LIN {X 0,Y 426.381,Z 386.373,A -85,B 0,C 180,E1 -9911.885,E2 -9911.885} C_VEL
LIN {X 0,Y 426.7,Z 374.582,A -85,B 0,C 180,E1 -9912.449,E2 -9912.449} C_VEL
LIN {X 0,Y 426.837,Z 364.477,A -85,B 0,C 180,E1 -9912.777,E2 -9912.777} C_VEL
LIN {X 0,Y 427.571,Z 302.941,A -85,B 0,C 180,E1 -9914.039,E2 -9914.039} C_VEL
LIN {X 0,Y 425.288,Z 288.443,A -85,B 0,C 180,E1 -9914.407,E2 -9914.407} C_VEL
LIN {X 0,Y 425.647,Z 277.739,A -85,B 0,C 180,E1 -9917.284,E2 -9917.284} C_VEL
LIN {X 0,Y 425.385,Z 272.31,A -85,B 0,C 180,E1 -9918.851,E2 -9918.851} C_VEL
LIN {X 0,Y 425.275,Z 272.323,A -85,B 0,C 180,E1 -9922.333,E2 -9922.333} C_VEL
LIN {X 0,Y 425.247,Z 272.327,A -85,B 0,C 180,E1 -9925.442,E2 -9925.442} C_VEL
LIN {X 0,Y 425.282,Z 272.324,A -85,B 0,C 180,E1 -9928.852,E2 -9928.852} C_VEL
LIN {X 0,Y 425.243,Z 272.328,A -85,B 0,C 180,E1 -9931.921,E2 -9931.921} C_VEL
LIN {X 0,Y 425.274,Z 272.323,A -85,B 0,C 180,E1 -9935.33,E2 -9935.33} C_VEL
LIN {X 0,Y 425.253,Z 272.327,A -85,B 0,C 180,E1 -9938.895,E2 -9938.895} C_VEL
LIN {X 0,Y 425.252,Z 272.326,A -85,B 0,C 180,E1 -9941.951,E2 -9941.951} C_VEL
LIN {X 0,Y 425.252,Z 272.328,A -85,B 0,C 180,E1 -9945.277,E2 -9945.277} C_VEL
LIN {X 0,Y 425.238,Z 272.327,A -85,B 0,C 180,E1 -9948.616,E2 -9948.616} C_VEL
LIN {X 0,Y 425.254,Z 272.326,A -85,B 0,C 180,E1 -9951.095,E2 -9951.095} C_VEL
LIN {X 0,Y 425.259,Z 272.325,A -85,B 0,C 180,E1 -9954.659,E2 -9954.659} C_VEL
LIN {X 0,Y 425.221,Z 272.329,A -85,B 0,C 180,E1 -9958.068,E2 -9958.068} C_VEL
LIN {X 0,Y 425.285,Z 272.322,A -85,B 0,C 180,E1 -9961.363,E2 -9961.363} C_VEL
LIN {X 0,Y 425.248,Z 272.327,A -85,B 0,C 180,E1 -9964.55,E2 -9964.55} C_VEL
LIN {X 0,Y 425.238,Z 272.328,A -85,B 0,C 180,E1 -9967.657,E2 -9967.657} C_VEL
LIN {X 0,Y 425.31,Z 272.319,A -85,B 0,C 180,E1 -9970.7,E2 -9970.7} C_VEL
LIN {X 0,Y 425.335,Z 272.316,A -85,B 0,C 180,E1 -9973.685,E2 -9973.685} C_VEL
LIN {X 0,Y 425.377,Z 272.31,A -85,B 0,C 180,E1 -9977.596,E2 -9977.596} C_VEL
LIN {X 0,Y 425.387,Z 272.309,A -85,B 0,C 180,E1 -9981.447,E2 -9981.447} C_VEL
LIN {X 0,Y 425.52,Z 272.295,A -85,B 0,C 180,E1 -9984.311,E2 -9984.311} C_VEL
LIN {X 0,Y 425.334,Z 272.315,A -85,B 0,C 180,E1 -9986.427,E2 -9986.427} C_VEL
LIN {X 0,Y 424.809,Z 272.381,A -85,B 0,C 180,E1 -9987.218,E2 -9987.218} C_VEL
LIN {X 0,Y 422.102,Z 272.72,A -85,B 0,C 180,E1 -9988.506,E2 -9988.506} C_VEL
LIN {X 0,Y 419.705,Z 273.017,A -85,B 0,C 180,E1 -9989.545,E2 -9989.545} C_VEL
LIN {X 0,Y 418.62,Z 273.153,A -85,B 0,C 180,E1 -9990.347,E2 -9990.347} C_VEL
LIN {X 0,Y 418.506,Z 273.164,A -85,B 0,C 180,E1 -9990.619,E2 -9990.619} C_VEL
LIN {X 0,Y 418.461,Z 273.172,A -85,B 0,C 180,E1 -9992.886,E2 -9992.886} C_VEL
LIN {X 0,Y 418.436,Z 273.176,A -85,B 0,C 180,E1 -9996.75,E2 -9996.75} C_VEL
LIN {X 0,Y 418.304,Z 273.192,A -85,B 0,C 180,E1 -9999.67,E2 -9999.67} C_VEL
LIN {X 0,Y 418.296,Z 273.193,A -85,B 0,C 180,E1 -10003.006,E2 -10003.006} C_VEL
LIN {X 0,Y 418.253,Z 273.199,A -85,B 0,C 180,E1 -10006.735,E2 -10006.735} C_VEL
LIN {X 0,Y 418.211,Z 273.203,A -85,B 0,C 180,E1 -10009.791,E2 -10009.791} C_VEL
LIN {X 0,Y 418.18,Z 273.207,A -85,B 0,C 180,E1 -10012.737,E2 -10012.737} C_VEL
LIN {X 0,Y 418.216,Z 273.202,A -85,B 0,C 180,E1 -10015.905,E2 -10015.905} C_VEL
LIN {X 0,Y 418.218,Z 273.204,A -85,B 0,C 180,E1 -10019.163,E2 -10019.163} C_VEL
LIN {X 0,Y 418.202,Z 273.204,A -85,B 0,C 180,E1 -10022.846,E2 -10022.846} C_VEL
LIN {X 0,Y 418.195,Z 273.205,A -85,B 0,C 180,E1 -10026.241,E2 -10026.241} C_VEL
LIN {X 0,Y 418.217,Z 273.203,A -85,B 0,C 180,E1 -10029.683,E2 -10029.683} C_VEL
LIN {X 0,Y 418.235,Z 273.2,A -85,B 0,C 180,E1 -10032.333,E2 -10032.333} C_VEL
LIN {X 0,Y 418.226,Z 273.201,A -85,B 0,C 180,E1 -10035.117,E2 -10035.117} C_VEL
LIN {X 0,Y 418.246,Z 273.201,A -85,B 0,C 180,E1 -10037.777,E2 -10037.777} C_VEL
LIN {X 0,Y 418.221,Z 273.202,A -85,B 0,C 180,E1 -10041.564,E2 -10041.564} C_VEL
LIN {X 0,Y 418.218,Z 273.202,A -85,B 0,C 180,E1 -10045.163,E2 -10045.163} C_VEL
LIN {X 0,Y 418.205,Z 273.203,A -85,B 0,C 180,E1 -10047.476,E2 -10047.476} C_VEL
LIN {X 0,Y 418.231,Z 273.2,A -85,B 0,C 180,E1 -10050.9,E2 -10050.9} C_VEL
LIN {X 0,Y 418.225,Z 273.203,A -85,B 0,C 180,E1 -10054.1,E2 -10054.1} C_VEL
LIN {X 0,Y 418.198,Z 273.205,A -85,B 0,C 180,E1 -10057.268,E2 -10057.268} C_VEL
LIN {X 0,Y 418.252,Z 273.2,A -85,B 0,C 180,E1 -10060.369,E2 -10060.369} C_VEL
LIN {X 0,Y 418.287,Z 273.194,A -85,B 0,C 180,E1 -10063.409,E2 -10063.409} C_VEL
LIN {X 0,Y 418.32,Z 273.189,A -85,B 0,C 180,E1 -10067.004,E2 -10067.004} C_VEL
LIN {X 0,Y 418.313,Z 273.191,A -85,B 0,C 180,E1 -10070.333,E2 -10070.333} C_VEL
LIN {X 0,Y 418.446,Z 273.173,A -85,B 0,C 180,E1 -10073.253,E2 -10073.253} C_VEL
LIN {X 0,Y 418.303,Z 273.191,A -85,B 0,C 180,E1 -10075.186,E2 -10075.186} C_VEL
LIN {X 0,Y 418.516,Z 273.165,A -85,B 0,C 180,E1 -10078.08,E2 -10078.08} C_VEL
LIN {X 0,Y 418.526,Z 273.164,A -85,B 0,C 180,E1 -10080.005,E2 -10080.005} C_VEL
LIN {X 0,Y 418.474,Z 273.172,A -85,B 0,C 180,E1 -10082.893,E2 -10082.893} C_VEL
LIN {X 0,Y 418.473,Z 273.17,A -85,B 0,C 180,E1 -10085.788,E2 -10085.788} C_VEL
LIN {X 0,Y 418.364,Z 273.184,A -85,B 0,C 180,E1 -10088.7,E2 -10088.7} C_VEL
LIN {X 0,Y 418.302,Z 273.191,A -85,B 0,C 180,E1 -10091.636,E2 -10091.636} C_VEL
LIN {X 0,Y 418.268,Z 273.196,A -85,B 0,C 180,E1 -10094.602,E2 -10094.602} C_VEL
LIN {X 0,Y 418.247,Z 273.199,A -85,B 0,C 180,E1 -10097.61,E2 -10097.61} C_VEL
LIN {X 0,Y 418.242,Z 273.199,A -85,B 0,C 180,E1 -10100.667,E2 -10100.667} C_VEL
LIN {X 0,Y 418.25,Z 273.199,A -85,B 0,C 180,E1 -10103.787,E2 -10103.787} C_VEL
LIN {X 0,Y 418.219,Z 273.202,A -85,B 0,C 180,E1 -10107.051,E2 -10107.051} C_VEL
LIN {X 0,Y 418.238,Z 273.199,A -85,B 0,C 180,E1 -10110.276,E2 -10110.276} C_VEL
LIN {X 0,Y 418.229,Z 273.202,A -85,B 0,C 180,E1 -10113.683,E2 -10113.683} C_VEL
LIN {X 0,Y 418.231,Z 273.2,A -85,B 0,C 180,E1 -10117.229,E2 -10117.229} C_VEL
LIN {X 0,Y 418.206,Z 273.203,A -85,B 0,C 180,E1 -10120.87,E2 -10120.87} C_VEL
LIN {X 0,Y 418.202,Z 273.204,A -85,B 0,C 180,E1 -10123.731,E2 -10123.731} C_VEL
LIN {X 0,Y 418.198,Z 273.205,A -85,B 0,C 180,E1 -10126.45,E2 -10126.45} C_VEL
LIN {X 0,Y 418.208,Z 273.203,A -85,B 0,C 180,E1 -10129.136,E2 -10129.136} C_VEL
LIN {X 0,Y 418.238,Z 273.199,A -85,B 0,C 180,E1 -10132.778,E2 -10132.778} C_VEL
LIN {X 0,Y 418.235,Z 273.202,A -85,B 0,C 180,E1 -10136.324,E2 -10136.324} C_VEL
LIN {X 0,Y 418.242,Z 273.199,A -85,B 0,C 180,E1 -10139.73,E2 -10139.73} C_VEL
LIN {X 0,Y 418.205,Z 273.203,A -85,B 0,C 180,E1 -10143.018,E2 -10143.018} C_VEL
LIN {X 0,Y 418.321,Z 273.357,A -85,B 0,C 180,E1 -10144.988,E2 -10144.988} C_VEL
LIN {X 0,Y 419.897,Z 283.23,A -85,B 0,C 180,E1 -10147.361,E2 -10147.361} C_VEL
LIN {X 0,Y 419.321,Z 295.276,A -85,B 0,C 180,E1 -10150.104,E2 -10150.104} C_VEL
LIN {X 0,Y 418.425,Z 312.199,A -85,B 0,C 180,E1 -10153.912,E2 -10153.912} C_VEL
LIN {X 0,Y 418.146,Z 318.839,A -85,B 0,C 180,E1 -10155.399,E2 -10155.399} C_VEL
LIN {X 0,Y 420.457,Z 340.768,A -85,B 0,C 180,E1 -10155.935,E2 -10155.935} C_VEL
LIN {X 0,Y 419.749,Z 397.826,A -85,B 0,C 180,E1 -10157.153,E2 -10157.153} C_VEL
LIN {X 0,Y 419.378,Z 409.923,A -85,B 0,C 180,E1 -10157.603,E2 -10157.603} C_VEL
LIN {X 0,Y 418.995,Z 419.778,A -85,B 0,C 180,E1 -10158.145,E2 -10158.145} C_VEL
LIN {X 0,Y 418.642,Z 428.317,A -85,B 0,C 180,E1 -10158.748,E2 -10158.748} C_VEL
LIN {X 0,Y 418.327,Z 436.579,A -85,B 0,C 180,E1 -10159.475,E2 -10159.475} C_VEL
LIN {X 0,Y 418.04,Z 444.456,A -85,B 0,C 180,E1 -10160.323,E2 -10160.323} C_VEL
LIN {X 0,Y 417.61,Z 453.524,A -85,B 0,C 180,E1 -10161.534,E2 -10161.534} C_VEL
LIN {X 0,Y 417.386,Z 460.516,A -85,B 0,C 180,E1 -10162.747,E2 -10162.747} C_VEL
LIN {X 0,Y 417.15,Z 466.408,A -85,B 0,C 180,E1 -10164.037,E2 -10164.037} C_VEL
LIN {X 0,Y 417.164,Z 470.478,A -85,B 0,C 180,E1 -10165.17,E2 -10165.17} C_VEL
LIN {X 0,Y 417.047,Z 473.209,A -85,B 0,C 180,E1 -10166.137,E2 -10166.137} C_VEL
LIN {X 0,Y 417.079,Z 475.349,A -85,B 0,C 180,E1 -10167.104,E2 -10167.104} C_VEL
LIN {X 0,Y 417.078,Z 476.927,A -85,B 0,C 180,E1 -10168.07,E2 -10168.07} C_VEL
LIN {X 0,Y 417.036,Z 477.901,A -85,B 0,C 180,E1 -10169.036,E2 -10169.036} C_VEL
LIN {X 0,Y 417.031,Z 478.279,A -85,B 0,C 180,E1 -10170.002,E2 -10170.002} C_VEL
LIN {X 0,Y 417.017,Z 478.147,A -85,B 0,C 180,E1 -10170.967,E2 -10170.967} C_VEL
LIN {X 0,Y 417.075,Z 477.507,A -85,B 0,C 180,E1 -10171.933,E2 -10171.933} C_VEL
LIN {X 0,Y 417.042,Z 476.345,A -85,B 0,C 180,E1 -10172.899,E2 -10172.899} C_VEL
LIN {X 0,Y 417.087,Z 473.43,A -85,B 0,C 180,E1 -10174.35,E2 -10174.35} C_VEL
LIN {X 0,Y 417.179,Z 469.185,A -85,B 0,C 180,E1 -10175.803,E2 -10175.803} C_VEL
LIN {X 0,Y 417.447,Z 463.483,A -85,B 0,C 180,E1 -10177.256,E2 -10177.256} C_VEL
LIN {X 0,Y 417.721,Z 457.262,A -85,B 0,C 180,E1 -10178.467,E2 -10178.467} C_VEL
LIN {X 0,Y 418.11,Z 451.182,A -85,B 0,C 180,E1 -10179.434,E2 -10179.434} C_VEL
LIN {X 0,Y 418.569,Z 443.809,A -85,B 0,C 180,E1 -10180.4,E2 -10180.4} C_VEL
LIN {X 0,Y 418.977,Z 435.985,A -85,B 0,C 180,E1 -10181.246,E2 -10181.246} C_VEL
LIN {X 0,Y 419.352,Z 429.321,A -85,B 0,C 180,E1 -10181.849,E2 -10181.849} C_VEL
LIN {X 0,Y 419.749,Z 421.293,A -85,B 0,C 180,E1 -10182.45,E2 -10182.45} C_VEL
LIN {X 0,Y 420.179,Z 412.209,A -85,B 0,C 180,E1 -10182.99,E2 -10182.99} C_VEL
LIN {X 0,Y 420.662,Z 402.136,A -85,B 0,C 180,E1 -10183.436,E2 -10183.436} C_VEL
LIN {X 0,Y 421.087,Z 390.096,A -85,B 0,C 180,E1 -10183.789,E2 -10183.789} C_VEL
LIN {X 0,Y 421.982,Z 339.107,A -85,B 0,C 180,E1 -10184.931,E2 -10184.931} C_VEL
LIN {X 0,Y 420.236,Z 325.232,A -85,B 0,C 180,E1 -10185.362,E2 -10185.362} C_VEL
LIN {X 0,Y 418.562,Z 315.696,A -85,B 0,C 180,E1 -10185.71,E2 -10185.71} C_VEL
LIN {X 0,Y 419.082,Z 299.8,A -85,B 0,C 180,E1 -10188.835,E2 -10188.835} C_VEL
LIN {X 0,Y 419.665,Z 282.928,A -85,B 0,C 180,E1 -10192.137,E2 -10192.137} C_VEL
LIN {X 0,Y 419.287,Z 277.639,A -85,B 0,C 180,E1 -10193.214,E2 -10193.214} C_VEL
LIN {X 0,Y 418.303,Z 273.195,A -85,B 0,C 180,E1 -10194.177,E2 -10194.177} C_VEL
LIN {X 0,Y 418.212,Z 273.208,A -85,B 0,C 180,E1 -10198.07,E2 -10198.07} C_VEL
LIN {X 0,Y 418.221,Z 273.206,A -85,B 0,C 180,E1 -10201.011,E2 -10201.011} C_VEL
LIN {X 0,Y 418.205,Z 273.204,A -85,B 0,C 180,E1 -10203.682,E2 -10203.682} C_VEL
LIN {X 0,Y 418.238,Z 273.201,A -85,B 0,C 180,E1 -10207.226,E2 -10207.226} C_VEL
LIN {X 0,Y 418.222,Z 273.205,A -85,B 0,C 180,E1 -10210.949,E2 -10210.949} C_VEL
LIN {X 0,Y 418.195,Z 273.202,A -85,B 0,C 180,E1 -10213.724,E2 -10213.724} C_VEL
LIN {X 0,Y 418.193,Z 273.203,A -85,B 0,C 180,E1 -10216.443,E2 -10216.443} C_VEL
LIN {X 0,Y 418.224,Z 273.201,A -85,B 0,C 180,E1 -10219.132,E2 -10219.132} C_VEL
LIN {X 0,Y 418.253,Z 273.197,A -85,B 0,C 180,E1 -10222.774,E2 -10222.774} C_VEL
LIN {X 0,Y 418.249,Z 273.196,A -85,B 0,C 180,E1 -10226.319,E2 -10226.319} C_VEL
LIN {X 0,Y 418.258,Z 273.198,A -85,B 0,C 180,E1 -10229.725,E2 -10229.725} C_VEL
LIN {X 0,Y 418.24,Z 273.204,A -85,B 0,C 180,E1 -10233.015,E2 -10233.015} C_VEL
LIN {X 0,Y 418.289,Z 273.196,A -85,B 0,C 180,E1 -10236.215,E2 -10236.215} C_VEL
LIN {X 0,Y 418.265,Z 273.199,A -85,B 0,C 180,E1 -10239.334,E2 -10239.334} C_VEL
LIN {X 0,Y 418.401,Z 273.384,A -85,B 0,C 180,E1 -10242.145,E2 -10242.145} C_VEL
LIN {X 0,Y 419.951,Z 279.942,A -85,B 0,C 180,E1 -10243.28,E2 -10243.28} C_VEL
LIN {X 0,Y 419.768,Z 287.188,A -85,B 0,C 180,E1 -10244.38,E2 -10244.38} C_VEL
LIN {X 0,Y 422.411,Z 302.684,A -85,B 0,C 180,E1 -10244.912,E2 -10244.912} C_VEL
LIN {X 0,Y 421.611,Z 349.13,A -85,B 0,C 180,E1 -10245.985,E2 -10245.985} C_VEL
LIN {X 0,Y 421.112,Z 370.004,A -85,B 0,C 180,E1 -10246.484,E2 -10246.484} C_VEL
LIN {X 0,Y 420.721,Z 381.477,A -85,B 0,C 180,E1 -10246.963,E2 -10246.963} C_VEL
LIN {X 0,Y 420.384,Z 389.953,A -85,B 0,C 180,E1 -10247.443,E2 -10247.443} C_VEL
LIN {X 0,Y 420.045,Z 398.323,A -85,B 0,C 180,E1 -10248.046,E2 -10248.046} C_VEL
LIN {X 0,Y 419.546,Z 406.458,A -85,B 0,C 180,E1 -10248.766,E2 -10248.766} C_VEL
LIN {X 0,Y 419.242,Z 414.199,A -85,B 0,C 180,E1 -10249.614,E2 -10249.614} C_VEL
LIN {X 0,Y 418.658,Z 423.145,A -85,B 0,C 180,E1 -10250.819,E2 -10250.819} C_VEL
LIN {X 0,Y 418.184,Z 430.047,A -85,B 0,C 180,E1 -10252.026,E2 -10252.026} C_VEL
LIN {X 0,Y 417.964,Z 435.543,A -85,B 0,C 180,E1 -10253.236,E2 -10253.236} C_VEL
LIN {X 0,Y 417.565,Z 439.126,A -85,B 0,C 180,E1 -10254.2,E2 -10254.2} C_VEL
LIN {X 0,Y 417.492,Z 443.184,A -85,B 0,C 180,E1 -10255.651,E2 -10255.651} C_VEL
LIN {X 0,Y 417.263,Z 445.971,A -85,B 0,C 180,E1 -10257.099,E2 -10257.099} C_VEL
LIN {X 0,Y 417.129,Z 447.063,A -85,B 0,C 180,E1 -10258.064,E2 -10258.064} C_VEL
LIN {X 0,Y 417.042,Z 447.644,A -85,B 0,C 180,E1 -10259.03,E2 -10259.03} C_VEL
LIN {X 0,Y 417.032,Z 447.72,A -85,B 0,C 180,E1 -10259.995,E2 -10259.995} C_VEL
LIN {X 0,Y 417.04,Z 447.28,A -85,B 0,C 180,E1 -10260.961,E2 -10260.961} C_VEL
LIN {X 0,Y 417.106,Z 446.234,A -85,B 0,C 180,E1 -10261.926,E2 -10261.926} C_VEL
LIN {X 0,Y 417.248,Z 443.672,A -85,B 0,C 180,E1 -10263.375,E2 -10263.375} C_VEL
LIN {X 0,Y 417.277,Z 439.705,A -85,B 0,C 180,E1 -10264.826,E2 -10264.826} C_VEL
LIN {X 0,Y 417.473,Z 434.89,A -85,B 0,C 180,E1 -10266.133,E2 -10266.133} C_VEL
LIN {X 0,Y 417.768,Z 428.599,A -85,B 0,C 180,E1 -10267.462,E2 -10267.462} C_VEL
LIN {X 0,Y 418.037,Z 421.038,A -85,B 0,C 180,E1 -10268.697,E2 -10268.697} C_VEL
LIN {X 0,Y 418.34,Z 413.649,A -85,B 0,C 180,E1 -10269.666,E2 -10269.666} C_VEL
LIN {X 0,Y 418.69,Z 405.785,A -85,B 0,C 180,E1 -10270.512,E2 -10270.512} C_VEL
LIN {X 0,Y 418.944,Z 397.53,A -85,B 0,C 180,E1 -10271.24,E2 -10271.24} C_VEL
LIN {X 0,Y 419.335,Z 387.148,A -85,B 0,C 180,E1 -10271.965,E2 -10271.965} C_VEL
LIN {X 0,Y 419.663,Z 375.717,A -85,B 0,C 180,E1 -10272.538,E2 -10272.538} C_VEL
LIN {X 0,Y 419.818,Z 366.071,A -85,B 0,C 180,E1 -10272.871,E2 -10272.871} C_VEL
LIN {X 0,Y 420.509,Z 303.025,A -85,B 0,C 180,E1 -10274.217,E2 -10274.217} C_VEL
LIN {X 0,Y 418.277,Z 288.664,A -85,B 0,C 180,E1 -10274.592,E2 -10274.592} C_VEL
LIN {X 0,Y 418.618,Z 277.685,A -85,B 0,C 180,E1 -10277.583,E2 -10277.583} C_VEL
LIN {X 0,Y 418.351,Z 273.186,A -85,B 0,C 180,E1 -10278.862,E2 -10278.862} C_VEL
LIN {X 0,Y 418.215,Z 273.203,A -85,B 0,C 180,E1 -10282.731,E2 -10282.731} C_VEL
LIN {X 0,Y 418.211,Z 273.203,A -85,B 0,C 180,E1 -10285.901,E2 -10285.901} C_VEL
LIN {X 0,Y 418.239,Z 273.199,A -85,B 0,C 180,E1 -10289.157,E2 -10289.157} C_VEL
LIN {X 0,Y 418.236,Z 273.202,A -85,B 0,C 180,E1 -10292.838,E2 -10292.838} C_VEL
LIN {X 0,Y 418.219,Z 273.202,A -85,B 0,C 180,E1 -10296.231,E2 -10296.231} C_VEL
LIN {X 0,Y 418.184,Z 273.206,A -85,B 0,C 180,E1 -10299.681,E2 -10299.681} C_VEL
LIN {X 0,Y 418.193,Z 273.206,A -85,B 0,C 180,E1 -10302.314,E2 -10302.314} C_VEL
LIN {X 0,Y 418.203,Z 273.205,A -85,B 0,C 180,E1 -10305.103,E2 -10305.103} C_VEL
LIN {X 0,Y 418.205,Z 273.203,A -85,B 0,C 180,E1 -10307.761,E2 -10307.761} C_VEL
LIN {X 0,Y 418.205,Z 273.204,A -85,B 0,C 180,E1 -10310.616,E2 -10310.616} C_VEL
LIN {X 0,Y 418.203,Z 273.203,A -85,B 0,C 180,E1 -10313.97,E2 -10313.97} C_VEL
LIN {X 0,Y 418.215,Z 273.202,A -85,B 0,C 180,E1 -10317.151,E2 -10317.151} C_VEL
LIN {X 0,Y 418.224,Z 273.202,A -85,B 0,C 180,E1 -10320.891,E2 -10320.891} C_VEL
LIN {X 0,Y 418.224,Z 273.201,A -85,B 0,C 180,E1 -10324.091,E2 -10324.091} C_VEL
LIN {X 0,Y 418.189,Z 273.206,A -85,B 0,C 180,E1 -10327.26,E2 -10327.26} C_VEL
LIN {X 0,Y 418.231,Z 273.2,A -85,B 0,C 180,E1 -10330.36,E2 -10330.36} C_VEL
LIN {X 0,Y 418.264,Z 273.196,A -85,B 0,C 180,E1 -10333.401,E2 -10333.401} C_VEL
LIN {X 0,Y 418.301,Z 273.192,A -85,B 0,C 180,E1 -10336.991,E2 -10336.991} C_VEL
LIN {X 0,Y 418.306,Z 273.192,A -85,B 0,C 180,E1 -10340.326,E2 -10340.326} C_VEL
LIN {X 0,Y 418.438,Z 273.176,A -85,B 0,C 180,E1 -10343.247,E2 -10343.247} C_VEL
LIN {X 0,Y 418.291,Z 273.193,A -85,B 0,C 180,E1 -10345.179,E2 -10345.179} C_VEL
LIN {X 0,Y 418.489,Z 273.169,A -85,B 0,C 180,E1 -10348.074,E2 -10348.074} C_VEL
LIN {X 0,Y 418.506,Z 273.164,A -85,B 0,C 180,E1 -10350.619,E2 -10350.619} C_VEL
LIN {X 0,Y 417.738,Z 273.263,A -85,B 0,C 180,E1 -10351.422,E2 -10351.422} C_VEL
LIN {X 0,Y 414.75,Z 273.634,A -85,B 0,C 180,E1 -10352.724,E2 -10352.724} C_VEL
LIN {X 0,Y 412.303,Z 273.939,A -85,B 0,C 180,E1 -10353.775,E2 -10353.775} C_VEL
LIN {X 0,Y 411.308,Z 274.064,A -85,B 0,C 180,E1 -10354.59,E2 -10354.59} C_VEL
LIN {X 0,Y 411.254,Z 274.069,A -85,B 0,C 180,E1 -10354.865,E2 -10354.865} C_VEL
LIN {X 0,Y 411.402,Z 274.051,A -85,B 0,C 180,E1 -10356.866,E2 -10356.866} C_VEL
LIN {X 0,Y 411.252,Z 274.071,A -85,B 0,C 180,E1 -10359.838,E2 -10359.838} C_VEL
LIN {X 0,Y 411.255,Z 274.069,A -85,B 0,C 180,E1 -10363.109,E2 -10363.109} C_VEL
LIN {X 0,Y 411.199,Z 274.078,A -85,B 0,C 180,E1 -10366.889,E2 -10366.889} C_VEL
LIN {X 0,Y 411.172,Z 274.08,A -85,B 0,C 180,E1 -10369.988,E2 -10369.988} C_VEL
LIN {X 0,Y 411.146,Z 274.084,A -85,B 0,C 180,E1 -10373.149,E2 -10373.149} C_VEL
LIN {X 0,Y 411.182,Z 274.079,A -85,B 0,C 180,E1 -10376.382,E2 -10376.382} C_VEL
LIN {X 0,Y 411.155,Z 274.081,A -85,B 0,C 180,E1 -10379.714,E2 -10379.714} C_VEL
LIN {X 0,Y 411.152,Z 274.083,A -85,B 0,C 180,E1 -10383.158,E2 -10383.158} C_VEL
LIN {X 0,Y 411.143,Z 274.084,A -85,B 0,C 180,E1 -10386.556,E2 -10386.556} C_VEL
LIN {X 0,Y 411.179,Z 274.079,A -85,B 0,C 180,E1 -10389.734,E2 -10389.734} C_VEL
LIN {X 0,Y 411.182,Z 274.079,A -85,B 0,C 180,E1 -10393.129,E2 -10393.129} C_VEL
LIN {X 0,Y 411.186,Z 274.078,A -85,B 0,C 180,E1 -10395.875,E2 -10395.875} C_VEL
LIN {X 0,Y 411.164,Z 274.081,A -85,B 0,C 180,E1 -10398.768,E2 -10398.768} C_VEL
LIN {X 0,Y 411.16,Z 274.082,A -85,B 0,C 180,E1 -10402.031,E2 -10402.031} C_VEL
LIN {X 0,Y 411.165,Z 274.081,A -85,B 0,C 180,E1 -10405.671,E2 -10405.671} C_VEL
LIN {X 0,Y 411.15,Z 274.083,A -85,B 0,C 180,E1 -10409.157,E2 -10409.157} C_VEL
LIN {X 0,Y 411.222,Z 274.073,A -85,B 0,C 180,E1 -10412.527,E2 -10412.527} C_VEL
LIN {X 0,Y 411.177,Z 274.079,A -85,B 0,C 180,E1 -10415.788,E2 -10415.788} C_VEL
LIN {X 0,Y 411.164,Z 274.08,A -85,B 0,C 180,E1 -10418.971,E2 -10418.971} C_VEL
LIN {X 0,Y 411.215,Z 274.075,A -85,B 0,C 180,E1 -10422.09,E2 -10422.09} C_VEL
LIN {X 0,Y 411.231,Z 274.072,A -85,B 0,C 180,E1 -10425.152,E2 -10425.152} C_VEL
LIN {X 0,Y 411.257,Z 274.069,A -85,B 0,C 180,E1 -10428.172,E2 -10428.172} C_VEL
LIN {X 0,Y 411.416,Z 274.049,A -85,B 0,C 180,E1 -10432.197,E2 -10432.197} C_VEL
LIN {X 0,Y 411.44,Z 274.046,A -85,B 0,C 180,E1 -10434.123,E2 -10434.123} C_VEL
LIN {X 0,Y 411.485,Z 274.041,A -85,B 0,C 180,E1 -10438.047,E2 -10438.047} C_VEL
LIN {X 0,Y 411.363,Z 274.058,A -85,B 0,C 180,E1 -10440.984,E2 -10440.984} C_VEL
LIN {X 0,Y 411.431,Z 274.05,A -85,B 0,C 180,E1 -10442.942,E2 -10442.942} C_VEL
LIN {X 0,Y 411.417,Z 274.049,A -85,B 0,C 180,E1 -10445.887,E2 -10445.887} C_VEL
LIN {X 0,Y 411.305,Z 274.064,A -85,B 0,C 180,E1 -10448.851,E2 -10448.851} C_VEL
LIN {X 0,Y 411.271,Z 274.067,A -85,B 0,C 180,E1 -10451.837,E2 -10451.837} C_VEL
LIN {X 0,Y 411.222,Z 274.074,A -85,B 0,C 180,E1 -10454.858,E2 -10454.858} C_VEL
LIN {X 0,Y 411.205,Z 274.075,A -85,B 0,C 180,E1 -10457.921,E2 -10457.921} C_VEL
LIN {X 0,Y 411.188,Z 274.078,A -85,B 0,C 180,E1 -10461.039,E2 -10461.039} C_VEL
LIN {X 0,Y 411.184,Z 274.077,A -85,B 0,C 180,E1 -10464.222,E2 -10464.222} C_VEL
LIN {X 0,Y 411.183,Z 274.08,A -85,B 0,C 180,E1 -10467.487,E2 -10467.487} C_VEL
LIN {X 0,Y 411.185,Z 274.079,A -85,B 0,C 180,E1 -10470.852,E2 -10470.852} C_VEL
LIN {X 0,Y 411.189,Z 274.077,A -85,B 0,C 180,E1 -10474.339,E2 -10474.339} C_VEL
LIN {X 0,Y 411.184,Z 274.078,A -85,B 0,C 180,E1 -10476.746,E2 -10476.746} C_VEL
LIN {X 0,Y 411.166,Z 274.081,A -85,B 0,C 180,E1 -10479.724,E2 -10479.724} C_VEL
LIN {X 0,Y 411.162,Z 274.082,A -85,B 0,C 180,E1 -10483.139,E2 -10483.139} C_VEL
LIN {X 0,Y 411.163,Z 274.082,A -85,B 0,C 180,E1 -10485.885,E2 -10485.885} C_VEL
LIN {X 0,Y 411.159,Z 274.081,A -85,B 0,C 180,E1 -10489.496,E2 -10489.496} C_VEL
LIN {X 0,Y 411.186,Z 274.079,A -85,B 0,C 180,E1 -10492.028,E2 -10492.028} C_VEL
LIN {X 0,Y 411.205,Z 274.075,A -85,B 0,C 180,E1 -10495.127,E2 -10495.127} C_VEL
LIN {X 0,Y 411.166,Z 274.08,A -85,B 0,C 180,E1 -10498.005,E2 -10498.005} C_VEL
LIN {X 0,Y 411.173,Z 274.079,A -85,B 0,C 180,E1 -10501.409,E2 -10501.409} C_VEL
LIN {X 0,Y 411.304,Z 274.259,A -85,B 0,C 180,E1 -10504.871,E2 -10504.871} C_VEL
LIN {X 0,Y 412.872,Z 283.842,A -85,B 0,C 180,E1 -10507.218,E2 -10507.218} C_VEL
LIN {X 0,Y 412.386,Z 294.15,A -85,B 0,C 180,E1 -10509.612,E2 -10509.612} C_VEL
LIN {X 0,Y 411.468,Z 310.565,A -85,B 0,C 180,E1 -10513.378,E2 -10513.378} C_VEL
LIN {X 0,Y 411.086,Z 318.732,A -85,B 0,C 180,E1 -10515.229,E2 -10515.229} C_VEL
LIN {X 0,Y 413.475,Z 340.317,A -85,B 0,C 180,E1 -10515.767,E2 -10515.767} C_VEL
LIN {X 0,Y 412.744,Z 396.594,A -85,B 0,C 180,E1 -10516.994,E2 -10516.994} C_VEL
LIN {X 0,Y 412.397,Z 407.766,A -85,B 0,C 180,E1 -10517.39,E2 -10517.39} C_VEL
LIN {X 0,Y 412.007,Z 418.175,A -85,B 0,C 180,E1 -10517.94,E2 -10517.94} C_VEL
LIN {X 0,Y 411.57,Z 428.466,A -85,B 0,C 180,E1 -10518.677,E2 -10518.677} C_VEL
LIN {X 0,Y 411.249,Z 436.658,A -85,B 0,C 180,E1 -10519.416,E2 -10519.416} C_VEL
LIN {X 0,Y 410.963,Z 444.487,A -85,B 0,C 180,E1 -10520.279,E2 -10520.279} C_VEL
LIN {X 0,Y 410.572,Z 452.694,A -85,B 0,C 180,E1 -10521.388,E2 -10521.388} C_VEL
LIN {X 0,Y 410.316,Z 459.83,A -85,B 0,C 180,E1 -10522.621,E2 -10522.621} C_VEL
LIN {X 0,Y 410.157,Z 464.65,A -85,B 0,C 180,E1 -10523.644,E2 -10523.644} C_VEL
LIN {X 0,Y 410.09,Z 468.376,A -85,B 0,C 180,E1 -10524.593,E2 -10524.593} C_VEL
LIN {X 0,Y 410.02,Z 471.51,A -85,B 0,C 180,E1 -10525.578,E2 -10525.578} C_VEL
LIN {X 0,Y 409.978,Z 474.946,A -85,B 0,C 180,E1 -10527.054,E2 -10527.054} C_VEL
LIN {X 0,Y 410.007,Z 476.568,A -85,B 0,C 180,E1 -10528.037,E2 -10528.037} C_VEL
LIN {X 0,Y 409.96,Z 477.557,A -85,B 0,C 180,E1 -10529.019,E2 -10529.019} C_VEL
LIN {X 0,Y 409.952,Z 477.981,A -85,B 0,C 180,E1 -10530.002,E2 -10530.002} C_VEL
LIN {X 0,Y 409.943,Z 477.892,A -85,B 0,C 180,E1 -10530.984,E2 -10530.984} C_VEL
LIN {X 0,Y 409.985,Z 477.293,A -85,B 0,C 180,E1 -10531.966,E2 -10531.966} C_VEL
LIN {X 0,Y 409.94,Z 476.165,A -85,B 0,C 180,E1 -10532.95,E2 -10532.95} C_VEL
LIN {X 0,Y 410.018,Z 473.305,A -85,B 0,C 180,E1 -10534.425,E2 -10534.425} C_VEL
LIN {X 0,Y 410.106,Z 470.732,A -85,B 0,C 180,E1 -10535.41,E2 -10535.41} C_VEL
LIN {X 0,Y 410.224,Z 466.581,A -85,B 0,C 180,E1 -10536.627,E2 -10536.627} C_VEL
LIN {X 0,Y 410.484,Z 461.148,A -85,B 0,C 180,E1 -10537.874,E2 -10537.874} C_VEL
LIN {X 0,Y 410.763,Z 455.908,A -85,B 0,C 180,E1 -10538.86,E2 -10538.86} C_VEL
LIN {X 0,Y 411.227,Z 449.607,A -85,B 0,C 180,E1 -10539.842,E2 -10539.842} C_VEL
LIN {X 0,Y 411.713,Z 441.967,A -85,B 0,C 180,E1 -10540.824,E2 -10540.824} C_VEL
LIN {X 0,Y 412.146,Z 433.828,A -85,B 0,C 180,E1 -10541.684,E2 -10541.684} C_VEL
LIN {X 0,Y 412.765,Z 423.769,A -85,B 0,C 180,E1 -10542.54,E2 -10542.54} C_VEL
LIN {X 0,Y 413.337,Z 413.26,A -85,B 0,C 180,E1 -10543.209,E2 -10543.209} C_VEL
LIN {X 0,Y 413.862,Z 402.988,A -85,B 0,C 180,E1 -10543.692,E2 -10543.692} C_VEL
LIN {X 0,Y 414.278,Z 393.279,A -85,B 0,C 180,E1 -10544.009,E2 -10544.009} C_VEL
LIN {X 0,Y 415.275,Z 339.307,A -85,B 0,C 180,E1 -10545.273,E2 -10545.273} C_VEL
LIN {X 0,Y 413.625,Z 326.463,A -85,B 0,C 180,E1 -10545.686,E2 -10545.686} C_VEL
LIN {X 0,Y 411.66,Z 315.383,A -85,B 0,C 180,E1 -10546.108,E2 -10546.108} C_VEL
LIN {X 0,Y 412.202,Z 300.045,A -85,B 0,C 180,E1 -10549.162,E2 -10549.162} C_VEL
LIN {X 0,Y 412.816,Z 284.495,A -85,B 0,C 180,E1 -10552.261,E2 -10552.261} C_VEL
LIN {X 0,Y 412.45,Z 279.407,A -85,B 0,C 180,E1 -10553.314,E2 -10553.314} C_VEL
LIN {X 0,Y 411.23,Z 274.076,A -85,B 0,C 180,E1 -10554.523,E2 -10554.523} C_VEL
LIN {X 0,Y 411.154,Z 274.088,A -85,B 0,C 180,E1 -10557.487,E2 -10557.487} C_VEL
LIN {X 0,Y 411.199,Z 274.079,A -85,B 0,C 180,E1 -10559.714,E2 -10559.714} C_VEL
LIN {X 0,Y 411.149,Z 274.084,A -85,B 0,C 180,E1 -10563.162,E2 -10563.162} C_VEL
LIN {X 0,Y 411.185,Z 274.079,A -85,B 0,C 180,E1 -10566.744,E2 -10566.744} C_VEL
LIN {X 0,Y 411.179,Z 274.075,A -85,B 0,C 180,E1 -10569.718,E2 -10569.718} C_VEL
LIN {X 0,Y 411.134,Z 274.085,A -85,B 0,C 180,E1 -10573.14,E2 -10573.14} C_VEL
LIN {X 0,Y 411.162,Z 274.077,A -85,B 0,C 180,E1 -10575.883,E2 -10575.883} C_VEL
LIN {X 0,Y 411.175,Z 274.075,A -85,B 0,C 180,E1 -10579.491,E2 -10579.491} C_VEL
LIN {X 0,Y 411.2,Z 274.071,A -85,B 0,C 180,E1 -10582.023,E2 -10582.023} C_VEL
LIN {X 0,Y 411.219,Z 274.074,A -85,B 0,C 180,E1 -10585.122,E2 -10585.122} C_VEL
LIN {X 0,Y 411.181,Z 274.078,A -85,B 0,C 180,E1 -10588,E2 -10588} C_VEL
LIN {X 0,Y 411.197,Z 274.081,A -85,B 0,C 180,E1 -10591.405,E2 -10591.405} C_VEL
LIN {X 0,Y 411.243,Z 274.076,A -85,B 0,C 180,E1 -10594.927,E2 -10594.927} C_VEL
LIN {X 0,Y 411.22,Z 274.077,A -85,B 0,C 180,E1 -10597.91,E2 -10597.91} C_VEL
LIN {X 0,Y 411.282,Z 274.069,A -85,B 0,C 180,E1 -10601.567,E2 -10601.567} C_VEL
LIN {X 0,Y 411.32,Z 274.247,A -85,B 0,C 180,E1 -10601.762,E2 -10601.762} C_VEL
LIN {X 0,Y 412.96,Z 280.42,A -85,B 0,C 180,E1 -10602.874,E2 -10602.874} C_VEL
LIN {X 0,Y 413.111,Z 283.875,A -85,B 0,C 180,E1 -10603.44,E2 -10603.44} C_VEL
LIN {X 0,Y 413.06,Z 287.577,A -85,B 0,C 180,E1 -10603.985,E2 -10603.985} C_VEL
LIN {X 0,Y 415.76,Z 303.008,A -85,B 0,C 180,E1 -10604.554,E2 -10604.554} C_VEL
LIN {X 0,Y 415.729,Z 313.745,A -85,B 0,C 180,E1 -10604.827,E2 -10604.827} C_VEL
LIN {X 0,Y 414.419,Z 369.033,A -85,B 0,C 180,E1 -10606.136,E2 -10606.136} C_VEL
LIN {X 0,Y 413.974,Z 381.064,A -85,B 0,C 180,E1 -10606.622,E2 -10606.622} C_VEL
LIN {X 0,Y 413.556,Z 391.414,A -85,B 0,C 180,E1 -10607.232,E2 -10607.232} C_VEL
LIN {X 0,Y 413.065,Z 400.988,A -85,B 0,C 180,E1 -10607.966,E2 -10607.966} C_VEL
LIN {X 0,Y 412.587,Z 410.969,A -85,B 0,C 180,E1 -10608.948,E2 -10608.948} C_VEL
LIN {X 0,Y 412.045,Z 418.812,A -85,B 0,C 180,E1 -10609.927,E2 -10609.927} C_VEL
LIN {X 0,Y 411.616,Z 425.292,A -85,B 0,C 180,E1 -10610.908,E2 -10610.908} C_VEL
LIN {X 0,Y 411.101,Z 431.874,A -85,B 0,C 180,E1 -10612.135,E2 -10612.135} C_VEL
LIN {X 0,Y 410.944,Z 436.128,A -85,B 0,C 180,E1 -10613.12,E2 -10613.12} C_VEL
LIN {X 0,Y 410.536,Z 439.656,A -85,B 0,C 180,E1 -10614.1,E2 -10614.1} C_VEL
LIN {X 0,Y 410.394,Z 442.505,A -85,B 0,C 180,E1 -10615.083,E2 -10615.083} C_VEL
LIN {X 0,Y 410.403,Z 444.749,A -85,B 0,C 180,E1 -10616.068,E2 -10616.068} C_VEL
LIN {X 0,Y 410.205,Z 446.387,A -85,B 0,C 180,E1 -10617.049,E2 -10617.049} C_VEL
LIN {X 0,Y 410.06,Z 447.425,A -85,B 0,C 180,E1 -10618.031,E2 -10618.031} C_VEL
LIN {X 0,Y 409.967,Z 447.949,A -85,B 0,C 180,E1 -10619.013,E2 -10619.013} C_VEL
LIN {X 0,Y 409.953,Z 447.968,A -85,B 0,C 180,E1 -10619.995,E2 -10619.995} C_VEL
LIN {X 0,Y 409.964,Z 447.486,A -85,B 0,C 180,E1 -10620.977,E2 -10620.977} C_VEL
LIN {X 0,Y 410.036,Z 446.423,A -85,B 0,C 180,E1 -10621.959,E2 -10621.959} C_VEL
LIN {X 0,Y 410.165,Z 443.756,A -85,B 0,C 180,E1 -10623.433,E2 -10623.433} C_VEL
LIN {X 0,Y 410.167,Z 441.279,A -85,B 0,C 180,E1 -10624.417,E2 -10624.417} C_VEL
LIN {X 0,Y 410.336,Z 436.221,A -85,B 0,C 180,E1 -10625.893,E2 -10625.893} C_VEL
LIN {X 0,Y 410.608,Z 430.76,A -85,B 0,C 180,E1 -10627.123,E2 -10627.123} C_VEL
LIN {X 0,Y 410.793,Z 425.391,A -85,B 0,C 180,E1 -10628.109,E2 -10628.109} C_VEL
LIN {X 0,Y 411.063,Z 418.92,A -85,B 0,C 180,E1 -10629.094,E2 -10629.094} C_VEL
LIN {X 0,Y 411.486,Z 410.016,A -85,B 0,C 180,E1 -10630.201,E2 -10630.201} C_VEL
LIN {X 0,Y 411.863,Z 399.711,A -85,B 0,C 180,E1 -10631.187,E2 -10631.187} C_VEL
LIN {X 0,Y 412.153,Z 391.628,A -85,B 0,C 180,E1 -10631.802,E2 -10631.802} C_VEL
LIN {X 0,Y 412.49,Z 382.438,A -85,B 0,C 180,E1 -10632.353,E2 -10632.353} C_VEL
LIN {X 0,Y 412.696,Z 372.919,A -85,B 0,C 180,E1 -10632.785,E2 -10632.785} C_VEL
LIN {X 0,Y 412.938,Z 361.942,A -85,B 0,C 180,E1 -10633.121,E2 -10633.121} C_VEL
LIN {X 0,Y 413.537,Z 303.984,A -85,B 0,C 180,E1 -10634.368,E2 -10634.368} C_VEL
LIN {X 0,Y 411.244,Z 288.92,A -85,B 0,C 180,E1 -10634.768,E2 -10634.768} C_VEL
LIN {X 0,Y 411.571,Z 277.618,A -85,B 0,C 180,E1 -10637.894,E2 -10637.894} C_VEL
LIN {X 0,Y 411.302,Z 274.064,A -85,B 0,C 180,E1 -10638.938,E2 -10638.938} C_VEL
LIN {X 0,Y 411.187,Z 274.079,A -85,B 0,C 180,E1 -10642.634,E2 -10642.634} C_VEL
LIN {X 0,Y 411.17,Z 274.079,A -85,B 0,C 180,E1 -10645.29,E2 -10645.29} C_VEL
LIN {X 0,Y 411.155,Z 274.083,A -85,B 0,C 180,E1 -10648.587,E2 -10648.587} C_VEL
LIN {X 0,Y 411.145,Z 274.084,A -85,B 0,C 180,E1 -10651.991,E2 -10651.991} C_VEL
LIN {X 0,Y 411.187,Z 274.08,A -85,B 0,C 180,E1 -10654.872,E2 -10654.872} C_VEL
LIN {X 0,Y 411.168,Z 274.081,A -85,B 0,C 180,E1 -10658.16,E2 -10658.16} C_VEL
LIN {X 0,Y 411.142,Z 274.083,A -85,B 0,C 180,E1 -10661.8,E2 -10661.8} C_VEL
LIN {X 0,Y 411.143,Z 274.083,A -85,B 0,C 180,E1 -10665.504,E2 -10665.504} C_VEL
LIN {X 0,Y 411.128,Z 274.085,A -85,B 0,C 180,E1 -10668.766,E2 -10668.766} C_VEL
LIN {X 0,Y 411.151,Z 274.082,A -85,B 0,C 180,E1 -10672.02,E2 -10672.02} C_VEL
LIN {X 0,Y 411.165,Z 274.081,A -85,B 0,C 180,E1 -10675.661,E2 -10675.661} C_VEL
LIN {X 0,Y 411.146,Z 274.083,A -85,B 0,C 180,E1 -10679.147,E2 -10679.147} C_VEL
LIN {X 0,Y 411.213,Z 274.074,A -85,B 0,C 180,E1 -10682.518,E2 -10682.518} C_VEL
LIN {X 0,Y 411.179,Z 274.081,A -85,B 0,C 180,E1 -10685.78,E2 -10685.78} C_VEL
LIN {X 0,Y 411.145,Z 274.084,A -85,B 0,C 180,E1 -10688.962,E2 -10688.962} C_VEL
LIN {X 0,Y 411.2,Z 274.077,A -85,B 0,C 180,E1 -10692.081,E2 -10692.081} C_VEL
LIN {X 0,Y 411.208,Z 274.076,A -85,B 0,C 180,E1 -10695.144,E2 -10695.144} C_VEL
LIN {X 0,Y 411.247,Z 274.072,A -85,B 0,C 180,E1 -10698.165,E2 -10698.165} C_VEL
LIN {X 0,Y 411.388,Z 274.055,A -85,B 0,C 180,E1 -10702.183,E2 -10702.183} C_VEL
LIN {X 0,Y 411.434,Z 274.048,A -85,B 0,C 180,E1 -10704.116,E2 -10704.116} C_VEL
LIN {X 0,Y 411.458,Z 274.044,A -85,B 0,C 180,E1 -10708.041,E2 -10708.041} C_VEL
LIN {X 0,Y 411.473,Z 274.04,A -85,B 0,C 180,E1 -10710.599,E2 -10710.599} C_VEL
LIN {X 0,Y 411.416,Z 274.049,A -85,B 0,C 180,E1 -10712.936,E2 -10712.936} C_VEL
LIN {X 0,Y 411.254,Z 274.069,A -85,B 0,C 180,E1 -10714.865,E2 -10714.865} C_VEL
LIN {X 0,Y 410.664,Z 274.147,A -85,B 0,C 180,E1 -10715.684,E2 -10715.684} C_VEL
LIN {X 0,Y 407.844,Z 274.5,A -85,B 0,C 180,E1 -10717.014,E2 -10717.014} C_VEL
LIN {X 0,Y 405.397,Z 274.802,A -85,B 0,C 180,E1 -10718.088,E2 -10718.088} C_VEL
LIN {X 0,Y 404.322,Z 274.933,A -85,B 0,C 180,E1 -10718.919,E2 -10718.919} C_VEL
LIN {X 0,Y 404.224,Z 274.944,A -85,B 0,C 180,E1 -10719.2,E2 -10719.2} C_VEL
LIN {X 0,Y 404.214,Z 274.947,A -85,B 0,C 180,E1 -10722.041,E2 -10722.041} C_VEL
LIN {X 0,Y 404.148,Z 274.954,A -85,B 0,C 180,E1 -10725.118,E2 -10725.118} C_VEL
LIN {X 0,Y 404.151,Z 274.955,A -85,B 0,C 180,E1 -10728.239,E2 -10728.239} C_VEL
LIN {X 0,Y 404.08,Z 274.962,A -85,B 0,C 180,E1 -10731.42,E2 -10731.42} C_VEL
LIN {X 0,Y 404.12,Z 274.958,A -85,B 0,C 180,E1 -10734.667,E2 -10734.667} C_VEL
LIN {X 0,Y 404.142,Z 274.955,A -85,B 0,C 180,E1 -10738.001,E2 -10738.001} C_VEL
LIN {X 0,Y 404.087,Z 274.962,A -85,B 0,C 180,E1 -10741.561,E2 -10741.561} C_VEL
LIN {X 0,Y 404.131,Z 274.957,A -85,B 0,C 180,E1 -10745.019,E2 -10745.019} C_VEL
LIN {X 0,Y 404.113,Z 274.96,A -85,B 0,C 180,E1 -10748.759,E2 -10748.759} C_VEL
LIN {X 0,Y 404.142,Z 274.957,A -85,B 0,C 180,E1 -10751.614,E2 -10751.614} C_VEL
LIN {X 0,Y 404.153,Z 274.954,A -85,B 0,C 180,E1 -10754.534,E2 -10754.534} C_VEL
LIN {X 0,Y 404.163,Z 274.953,A -85,B 0,C 180,E1 -10757.309,E2 -10757.309} C_VEL
LIN {X 0,Y 404.124,Z 274.958,A -85,B 0,C 180,E1 -10759.959,E2 -10759.959} C_VEL
LIN {X 0,Y 404.098,Z 274.961,A -85,B 0,C 180,E1 -10763.128,E2 -10763.128} C_VEL
LIN {X 0,Y 404.104,Z 274.96,A -85,B 0,C 180,E1 -10766.192,E2 -10766.192} C_VEL
LIN {X 0,Y 404.107,Z 274.96,A -85,B 0,C 180,E1 -10769.719,E2 -10769.719} C_VEL
LIN {X 0,Y 404.157,Z 274.954,A -85,B 0,C 180,E1 -10773.127,E2 -10773.127} C_VEL
LIN {X 0,Y 404.135,Z 274.957,A -85,B 0,C 180,E1 -10775.339,E2 -10775.339} C_VEL
LIN {X 0,Y 404.106,Z 274.96,A -85,B 0,C 180,E1 -10778.585,E2 -10778.585} C_VEL
LIN {X 0,Y 404.174,Z 274.952,A -85,B 0,C 180,E1 -10781.767,E2 -10781.767} C_VEL
LIN {X 0,Y 404.177,Z 274.95,A -85,B 0,C 180,E1 -10784.887,E2 -10784.887} C_VEL
LIN {X 0,Y 404.23,Z 274.945,A -85,B 0,C 180,E1 -10787.964,E2 -10787.964} C_VEL
LIN {X 0,Y 404.242,Z 274.942,A -85,B 0,C 180,E1 -10791.003,E2 -10791.003} C_VEL
LIN {X 0,Y 404.388,Z 274.925,A -85,B 0,C 180,E1 -10794.02,E2 -10794.02} C_VEL
LIN {X 0,Y 404.453,Z 274.917,A -85,B 0,C 180,E1 -10798.014,E2 -10798.014} C_VEL
LIN {X 0,Y 404.334,Z 274.933,A -85,B 0,C 180,E1 -10801.001,E2 -10801.001} C_VEL
LIN {X 0,Y 404.389,Z 274.926,A -85,B 0,C 180,E1 -10802.993,E2 -10802.993} C_VEL
LIN {X 0,Y 404.366,Z 274.927,A -85,B 0,C 180,E1 -10805.99,E2 -10805.99} C_VEL
LIN {X 0,Y 404.253,Z 274.943,A -85,B 0,C 180,E1 -10809.006,E2 -10809.006} C_VEL
LIN {X 0,Y 404.244,Z 274.942,A -85,B 0,C 180,E1 -10812.046,E2 -10812.046} C_VEL
LIN {X 0,Y 404.166,Z 274.954,A -85,B 0,C 180,E1 -10815.124,E2 -10815.124} C_VEL
LIN {X 0,Y 404.158,Z 274.953,A -85,B 0,C 180,E1 -10818.245,E2 -10818.245} C_VEL
LIN {X 0,Y 404.13,Z 274.959,A -85,B 0,C 180,E1 -10821.424,E2 -10821.424} C_VEL
LIN {X 0,Y 404.142,Z 274.956,A -85,B 0,C 180,E1 -10824.672,E2 -10824.672} C_VEL
LIN {X 0,Y 404.125,Z 274.957,A -85,B 0,C 180,E1 -10828.009,E2 -10828.009} C_VEL
LIN {X 0,Y 404.141,Z 274.955,A -85,B 0,C 180,E1 -10830.289,E2 -10830.289} C_VEL
LIN {X 0,Y 404.135,Z 274.958,A -85,B 0,C 180,E1 -10833.817,E2 -10833.817} C_VEL
LIN {X 0,Y 404.13,Z 274.957,A -85,B 0,C 180,E1 -10836.878,E2 -10836.878} C_VEL
LIN {X 0,Y 404.117,Z 274.96,A -85,B 0,C 180,E1 -10840.078,E2 -10840.078} C_VEL
LIN {X 0,Y 404.142,Z 274.956,A -85,B 0,C 180,E1 -10843.085,E2 -10843.085} C_VEL
LIN {X 0,Y 404.12,Z 274.959,A -85,B 0,C 180,E1 -10845.925,E2 -10845.925} C_VEL
LIN {X 0,Y 404.102,Z 274.96,A -85,B 0,C 180,E1 -10848.636,E2 -10848.636} C_VEL
LIN {X 0,Y 404.141,Z 274.956,A -85,B 0,C 180,E1 -10851.498,E2 -10851.498} C_VEL
LIN {X 0,Y 404.176,Z 274.95,A -85,B 0,C 180,E1 -10854.986,E2 -10854.986} C_VEL
LIN {X 0,Y 404.141,Z 274.958,A -85,B 0,C 180,E1 -10858.446,E2 -10858.446} C_VEL
LIN {X 0,Y 404.153,Z 274.954,A -85,B 0,C 180,E1 -10860.865,E2 -10860.865} C_VEL
LIN {X 0,Y 404.206,Z 274.955,A -85,B 0,C 180,E1 -10864.712,E2 -10864.712} C_VEL
LIN {X 0,Y 405.865,Z 284.782,A -85,B 0,C 180,E1 -10867.158,E2 -10867.158} C_VEL
LIN {X 0,Y 405.296,Z 295.595,A -85,B 0,C 180,E1 -10869.71,E2 -10869.71} C_VEL
LIN {X 0,Y 404.39,Z 311.249,A -85,B 0,C 180,E1 -10873.365,E2 -10873.365} C_VEL
LIN {X 0,Y 404.031,Z 318.449,A -85,B 0,C 180,E1 -10875.037,E2 -10875.037} C_VEL
LIN {X 0,Y 406.46,Z 341.821,A -85,B 0,C 180,E1 -10875.637,E2 -10875.637} C_VEL
LIN {X 0,Y 405.716,Z 396.493,A -85,B 0,C 180,E1 -10876.86,E2 -10876.86} C_VEL
LIN {X 0,Y 405.365,Z 408.307,A -85,B 0,C 180,E1 -10877.295,E2 -10877.295} C_VEL
LIN {X 0,Y 404.947,Z 418.423,A -85,B 0,C 180,E1 -10877.854,E2 -10877.854} C_VEL
LIN {X 0,Y 404.589,Z 427.117,A -85,B 0,C 180,E1 -10878.479,E2 -10878.479} C_VEL
LIN {X 0,Y 404.177,Z 435.488,A -85,B 0,C 180,E1 -10879.228,E2 -10879.228} C_VEL
LIN {X 0,Y 403.913,Z 442.428,A -85,B 0,C 180,E1 -10879.982,E2 -10879.982} C_VEL
LIN {X 0,Y 403.641,Z 448.323,A -85,B 0,C 180,E1 -10880.734,E2 -10880.734} C_VEL
LIN {X 0,Y 403.397,Z 454.902,A -85,B 0,C 180,E1 -10881.738,E2 -10881.738} C_VEL
LIN {X 0,Y 403.214,Z 460.358,A -85,B 0,C 180,E1 -10882.742,E2 -10882.742} C_VEL
LIN {X 0,Y 403.066,Z 464.59,A -85,B 0,C 180,E1 -10883.67,E2 -10883.67} C_VEL
LIN {X 0,Y 403.004,Z 469.422,A -85,B 0,C 180,E1 -10885,E2 -10885} C_VEL
LIN {X 0,Y 402.888,Z 472.279,A -85,B 0,C 180,E1 -10886.001,E2 -10886.001} C_VEL
LIN {X 0,Y 402.879,Z 474.533,A -85,B 0,C 180,E1 -10887.002,E2 -10887.002} C_VEL
LIN {X 0,Y 402.937,Z 476.185,A -85,B 0,C 180,E1 -10888.003,E2 -10888.003} C_VEL
LIN {X 0,Y 402.887,Z 477.197,A -85,B 0,C 180,E1 -10889.002,E2 -10889.002} C_VEL
LIN {X 0,Y 402.876,Z 477.676,A -85,B 0,C 180,E1 -10890.002,E2 -10890.002} C_VEL
LIN {X 0,Y 402.87,Z 477.643,A -85,B 0,C 180,E1 -10891.001,E2 -10891.001} C_VEL
LIN {X 0,Y 402.883,Z 477.098,A -85,B 0,C 180,E1 -10892.001,E2 -10892.001} C_VEL
LIN {X 0,Y 402.839,Z 475.997,A -85,B 0,C 180,E1 -10893.002,E2 -10893.002} C_VEL
LIN {X 0,Y 402.95,Z 473.213,A -85,B 0,C 180,E1 -10894.503,E2 -10894.503} C_VEL
LIN {X 0,Y 403.025,Z 470.678,A -85,B 0,C 180,E1 -10895.505,E2 -10895.505} C_VEL
LIN {X 0,Y 403.214,Z 465.516,A -85,B 0,C 180,E1 -10897.01,E2 -10897.01} C_VEL
LIN {X 0,Y 403.524,Z 459.966,A -85,B 0,C 180,E1 -10898.263,E2 -10898.263} C_VEL
LIN {X 0,Y 403.853,Z 454.542,A -85,B 0,C 180,E1 -10899.265,E2 -10899.265} C_VEL
LIN {X 0,Y 404.324,Z 448.069,A -85,B 0,C 180,E1 -10900.265,E2 -10900.265} C_VEL
LIN {X 0,Y 404.96,Z 439.191,A -85,B 0,C 180,E1 -10901.387,E2 -10901.387} C_VEL
LIN {X 0,Y 405.609,Z 429.02,A -85,B 0,C 180,E1 -10902.383,E2 -10902.383} C_VEL
LIN {X 0,Y 406.216,Z 419.292,A -85,B 0,C 180,E1 -10903.127,E2 -10903.127} C_VEL
LIN {X 0,Y 406.806,Z 408.796,A -85,B 0,C 180,E1 -10903.743,E2 -10903.743} C_VEL
LIN {X 0,Y 407.418,Z 396.708,A -85,B 0,C 180,E1 -10904.231,E2 -10904.231} C_VEL
LIN {X 0,Y 408.742,Z 340.888,A -85,B 0,C 180,E1 -10905.592,E2 -10905.592} C_VEL
LIN {X 0,Y 407.117,Z 327.757,A -85,B 0,C 180,E1 -10906.035,E2 -10906.035} C_VEL
LIN {X 0,Y 404.754,Z 314.898,A -85,B 0,C 180,E1 -10906.553,E2 -10906.553} C_VEL
LIN {X 0,Y 405.401,Z 299.079,A -85,B 0,C 180,E1 -10909.76,E2 -10909.76} C_VEL
LIN {X 0,Y 405.957,Z 285.005,A -85,B 0,C 180,E1 -10912.618,E2 -10912.618} C_VEL
LIN {X 0,Y 405.584,Z 280.933,A -85,B 0,C 180,E1 -10913.489,E2 -10913.489} C_VEL
LIN {X 0,Y 404.191,Z 274.953,A -85,B 0,C 180,E1 -10914.854,E2 -10914.854} C_VEL
LIN {X 0,Y 404.113,Z 274.965,A -85,B 0,C 180,E1 -10918.007,E2 -10918.007} C_VEL
LIN {X 0,Y 404.139,Z 274.96,A -85,B 0,C 180,E1 -10920.287,E2 -10920.287} C_VEL
LIN {X 0,Y 404.094,Z 274.961,A -85,B 0,C 180,E1 -10923.819,E2 -10923.819} C_VEL
LIN {X 0,Y 404.138,Z 274.955,A -85,B 0,C 180,E1 -10927.494,E2 -10927.494} C_VEL
LIN {X 0,Y 404.135,Z 274.953,A -85,B 0,C 180,E1 -10930.074,E2 -10930.074} C_VEL
LIN {X 0,Y 404.093,Z 274.963,A -85,B 0,C 180,E1 -10933.071,E2 -10933.071} C_VEL
LIN {X 0,Y 404.121,Z 274.954,A -85,B 0,C 180,E1 -10935.918,E2 -10935.918} C_VEL
LIN {X 0,Y 404.115,Z 274.957,A -85,B 0,C 180,E1 -10938.631,E2 -10938.631} C_VEL
LIN {X 0,Y 404.156,Z 274.95,A -85,B 0,C 180,E1 -10941.494,E2 -10941.494} C_VEL
LIN {X 0,Y 404.19,Z 274.951,A -85,B 0,C 180,E1 -10944.981,E2 -10944.981} C_VEL
LIN {X 0,Y 404.155,Z 274.954,A -85,B 0,C 180,E1 -10948.44,E2 -10948.44} C_VEL
LIN {X 0,Y 404.169,Z 274.954,A -85,B 0,C 180,E1 -10950.86,E2 -10950.86} C_VEL
LIN {X 0,Y 404.162,Z 274.956,A -85,B 0,C 180,E1 -10954.228,E2 -10954.228} C_VEL
LIN {X 0,Y 404.184,Z 274.955,A -85,B 0,C 180,E1 -10957.505,E2 -10957.505} C_VEL
LIN {X 0,Y 404.229,Z 274.948,A -85,B 0,C 180,E1 -10961.233,E2 -10961.233} C_VEL
LIN {X 0,Y 404.267,Z 275.265,A -85,B 0,C 180,E1 -10961.367,E2 -10961.367} C_VEL
LIN {X 0,Y 406.395,Z 283.552,A -85,B 0,C 180,E1 -10962.899,E2 -10962.899} C_VEL
LIN {X 0,Y 406.353,Z 287.812,A -85,B 0,C 180,E1 -10963.568,E2 -10963.568} C_VEL
LIN {X 0,Y 409.225,Z 303.678,A -85,B 0,C 180,E1 -10964.176,E2 -10964.176} C_VEL
LIN {X 0,Y 409.246,Z 312.708,A -85,B 0,C 180,E1 -10964.419,E2 -10964.419} C_VEL
LIN {X 0,Y 407.702,Z 370.172,A -85,B 0,C 180,E1 -10965.84,E2 -10965.84} C_VEL
LIN {X 0,Y 407.225,Z 381.806,A -85,B 0,C 180,E1 -10966.332,E2 -10966.332} C_VEL
LIN {X 0,Y 406.835,Z 391.159,A -85,B 0,C 180,E1 -10966.891,E2 -10966.891} C_VEL
LIN {X 0,Y 406.431,Z 399.371,A -85,B 0,C 180,E1 -10967.513,E2 -10967.513} C_VEL
LIN {X 0,Y 405.866,Z 407.399,A -85,B 0,C 180,E1 -10968.256,E2 -10968.256} C_VEL
LIN {X 0,Y 405.508,Z 415.048,A -85,B 0,C 180,E1 -10969.132,E2 -10969.132} C_VEL
LIN {X 0,Y 404.875,Z 423.122,A -85,B 0,C 180,E1 -10970.252,E2 -10970.252} C_VEL
LIN {X 0,Y 404.294,Z 430.175,A -85,B 0,C 180,E1 -10971.498,E2 -10971.498} C_VEL
LIN {X 0,Y 403.994,Z 435.663,A -85,B 0,C 180,E1 -10972.728,E2 -10972.728} C_VEL
LIN {X 0,Y 403.51,Z 440.185,A -85,B 0,C 180,E1 -10973.997,E2 -10973.997} C_VEL
LIN {X 0,Y 403.326,Z 442.984,A -85,B 0,C 180,E1 -10974.997,E2 -10974.997} C_VEL
LIN {X 0,Y 403.355,Z 445.176,A -85,B 0,C 180,E1 -10975.999,E2 -10975.999} C_VEL
LIN {X 0,Y 403.15,Z 446.798,A -85,B 0,C 180,E1 -10976.997,E2 -10976.997} C_VEL
LIN {X 0,Y 402.993,Z 447.796,A -85,B 0,C 180,E1 -10977.996,E2 -10977.996} C_VEL
LIN {X 0,Y 402.893,Z 448.259,A -85,B 0,C 180,E1 -10978.996,E2 -10978.996} C_VEL
LIN {X 0,Y 402.877,Z 448.215,A -85,B 0,C 180,E1 -10979.995,E2 -10979.995} C_VEL
LIN {X 0,Y 402.89,Z 447.668,A -85,B 0,C 180,E1 -10980.994,E2 -10980.994} C_VEL
LIN {X 0,Y 402.968,Z 446.577,A -85,B 0,C 180,E1 -10981.994,E2 -10981.994} C_VEL
LIN {X 0,Y 403.062,Z 443.79,A -85,B 0,C 180,E1 -10983.494,E2 -10983.494} C_VEL
LIN {X 0,Y 403.09,Z 441.264,A -85,B 0,C 180,E1 -10984.495,E2 -10984.495} C_VEL
LIN {X 0,Y 403.206,Z 438.049,A -85,B 0,C 180,E1 -10985.496,E2 -10985.496} C_VEL
LIN {X 0,Y 403.522,Z 431.764,A -85,B 0,C 180,E1 -10986.997,E2 -10986.997} C_VEL
LIN {X 0,Y 403.681,Z 426.543,A -85,B 0,C 180,E1 -10988.001,E2 -10988.001} C_VEL
LIN {X 0,Y 403.934,Z 420.242,A -85,B 0,C 180,E1 -10989.003,E2 -10989.003} C_VEL
LIN {X 0,Y 404.203,Z 413.633,A -85,B 0,C 180,E1 -10989.881,E2 -10989.881} C_VEL
LIN {X 0,Y 404.63,Z 405.669,A -85,B 0,C 180,E1 -10990.756,E2 -10990.756} C_VEL
LIN {X 0,Y 404.919,Z 397.291,A -85,B 0,C 180,E1 -10991.508,E2 -10991.508} C_VEL
LIN {X 0,Y 405.314,Z 386.717,A -85,B 0,C 180,E1 -10992.258,E2 -10992.258} C_VEL
LIN {X 0,Y 405.621,Z 375.57,A -85,B 0,C 180,E1 -10992.82,E2 -10992.82} C_VEL
LIN {X 0,Y 405.802,Z 365.772,A -85,B 0,C 180,E1 -10993.165,E2 -10993.165} C_VEL
LIN {X 0,Y 406.572,Z 304.787,A -85,B 0,C 180,E1 -10994.527,E2 -10994.527} C_VEL
LIN {X 0,Y 404.218,Z 289.124,A -85,B 0,C 180,E1 -10994.958,E2 -10994.958} C_VEL
LIN {X 0,Y 404.54,Z 279.353,A -85,B 0,C 180,E1 -10997.693,E2 -10997.693} C_VEL
LIN {X 0,Y 404.264,Z 274.94,A -85,B 0,C 180,E1 -10999.018,E2 -10999.018} C_VEL
LIN {X 0,Y 404.134,Z 274.956,A -85,B 0,C 180,E1 -11002.824,E2 -11002.824} C_VEL
LIN {X 0,Y 404.122,Z 274.959,A -85,B 0,C 180,E1 -11005.763,E2 -11005.763} C_VEL
LIN {X 0,Y 404.135,Z 274.956,A -85,B 0,C 180,E1 -11009.596,E2 -11009.596} C_VEL
LIN {X 0,Y 404.12,Z 274.959,A -85,B 0,C 180,E1 -11012.615,E2 -11012.615} C_VEL
LIN {X 0,Y 404.157,Z 274.953,A -85,B 0,C 180,E1 -11015.183,E2 -11015.183} C_VEL
LIN {X 0,Y 404.11,Z 274.96,A -85,B 0,C 180,E1 -11018.753,E2 -11018.753} C_VEL
LIN {X 0,Y 404.088,Z 274.961,A -85,B 0,C 180,E1 -11021.592,E2 -11021.592} C_VEL
LIN {X 0,Y 404.113,Z 274.96,A -85,B 0,C 180,E1 -11024.516,E2 -11024.516} C_VEL
LIN {X 0,Y 404.102,Z 274.962,A -85,B 0,C 180,E1 -11027.29,E2 -11027.29} C_VEL
LIN {X 0,Y 404.119,Z 274.957,A -85,B 0,C 180,E1 -11029.948,E2 -11029.948} C_VEL
LIN {X 0,Y 404.097,Z 274.962,A -85,B 0,C 180,E1 -11033.12,E2 -11033.12} C_VEL
LIN {X 0,Y 404.104,Z 274.959,A -85,B 0,C 180,E1 -11036.182,E2 -11036.182} C_VEL
LIN {X 0,Y 404.102,Z 274.961,A -85,B 0,C 180,E1 -11039.71,E2 -11039.71} C_VEL
LIN {X 0,Y 404.149,Z 274.955,A -85,B 0,C 180,E1 -11043.118,E2 -11043.118} C_VEL
LIN {X 0,Y 404.13,Z 274.957,A -85,B 0,C 180,E1 -11045.33,E2 -11045.33} C_VEL
LIN {X 0,Y 404.088,Z 274.961,A -85,B 0,C 180,E1 -11048.576,E2 -11048.576} C_VEL
LIN {X 0,Y 404.158,Z 274.955,A -85,B 0,C 180,E1 -11051.758,E2 -11051.758} C_VEL
LIN {X 0,Y 404.154,Z 274.954,A -85,B 0,C 180,E1 -11054.879,E2 -11054.879} C_VEL
LIN {X 0,Y 404.218,Z 274.948,A -85,B 0,C 180,E1 -11057.956,E2 -11057.956} C_VEL
LIN {X 0,Y 404.329,Z 274.933,A -85,B 0,C 180,E1 -11062.005,E2 -11062.005} C_VEL
LIN {X 0,Y 404.38,Z 274.927,A -85,B 0,C 180,E1 -11064.013,E2 -11064.013} C_VEL
LIN {X 0,Y 404.427,Z 274.92,A -85,B 0,C 180,E1 -11068.007,E2 -11068.007} C_VEL
LIN {X 0,Y 404.555,Z 274.904,A -85,B 0,C 180,E1 -11069.998,E2 -11069.998} C_VEL
LIN {X 0,Y 404.373,Z 274.926,A -85,B 0,C 180,E1 -11072.987,E2 -11072.987} C_VEL
LIN {X 0,Y 404.349,Z 274.929,A -85,B 0,C 180,E1 -11076.987,E2 -11076.987} C_VEL
LIN {X 0,Y 404.224,Z 274.944,A -85,B 0,C 180,E1 -11079.2,E2 -11079.2} C_VEL
LIN {X 0,Y 403.536,Z 275.032,A -85,B 0,C 180,E1 -11080.032,E2 -11080.032} C_VEL
LIN {X 0,Y 400.699,Z 275.383,A -85,B 0,C 180,E1 -11081.383,E2 -11081.383} C_VEL
LIN {X 0,Y 398.296,Z 275.685,A -85,B 0,C 180,E1 -11082.475,E2 -11082.475} C_VEL
LIN {X 0,Y 397.242,Z 275.814,A -85,B 0,C 180,E1 -11083.318,E2 -11083.318} C_VEL
LIN {X 0,Y 397.143,Z 275.825,A -85,B 0,C 180,E1 -11083.604,E2 -11083.604} C_VEL
LIN {X 0,Y 397.124,Z 275.829,A -85,B 0,C 180,E1 -11087.155,E2 -11087.155} C_VEL
LIN {X 0,Y 397.045,Z 275.841,A -85,B 0,C 180,E1 -11090.731,E2 -11090.731} C_VEL
LIN {X 0,Y 397.076,Z 275.835,A -85,B 0,C 180,E1 -11094.02,E2 -11094.02} C_VEL
LIN {X 0,Y 397.139,Z 275.828,A -85,B 0,C 180,E1 -11097.392,E2 -11097.392} C_VEL
LIN {X 0,Y 397.029,Z 275.842,A -85,B 0,C 180,E1 -11100.884,E2 -11100.884} C_VEL
LIN {X 0,Y 397.072,Z 275.837,A -85,B 0,C 180,E1 -11104.496,E2 -11104.496} C_VEL
LIN {X 0,Y 397.059,Z 275.837,A -85,B 0,C 180,E1 -11108.277,E2 -11108.277} C_VEL
LIN {X 0,Y 397.107,Z 275.831,A -85,B 0,C 180,E1 -11111.997,E2 -11111.997} C_VEL
LIN {X 0,Y 397.103,Z 275.833,A -85,B 0,C 180,E1 -11115.063,E2 -11115.063} C_VEL
LIN {X 0,Y 397.11,Z 275.831,A -85,B 0,C 180,E1 -11118.011,E2 -11118.011} C_VEL
LIN {X 0,Y 397.066,Z 275.839,A -85,B 0,C 180,E1 -11121.73,E2 -11121.73} C_VEL
LIN {X 0,Y 397.085,Z 275.835,A -85,B 0,C 180,E1 -11125.511,E2 -11125.511} C_VEL
LIN {X 0,Y 397.04,Z 275.841,A -85,B 0,C 180,E1 -11129.122,E2 -11129.122} C_VEL
LIN {X 0,Y 397.157,Z 275.824,A -85,B 0,C 180,E1 -11132.615,E2 -11132.615} C_VEL
LIN {X 0,Y 397.091,Z 275.835,A -85,B 0,C 180,E1 -11135.986,E2 -11135.986} C_VEL
LIN {X 0,Y 397.108,Z 275.832,A -85,B 0,C 180,E1 -11139.71,E2 -11139.71} C_VEL
LIN {X 0,Y 397.153,Z 275.825,A -85,B 0,C 180,E1 -11142.85,E2 -11142.85} C_VEL
LIN {X 0,Y 397.203,Z 275.82,A -85,B 0,C 180,E1 -11146.708,E2 -11146.708} C_VEL
LIN {X 0,Y 397.191,Z 275.822,A -85,B 0,C 180,E1 -11149.814,E2 -11149.814} C_VEL
LIN {X 0,Y 397.309,Z 275.807,A -85,B 0,C 180,E1 -11152.893,E2 -11152.893} C_VEL
LIN {X 0,Y 397.221,Z 275.818,A -85,B 0,C 180,E1 -11154.93,E2 -11154.93} C_VEL
LIN {X 0,Y 397.422,Z 275.794,A -85,B 0,C 180,E1 -11157.978,E2 -11157.978} C_VEL
LIN {X 0,Y 397.304,Z 275.808,A -85,B 0,C 180,E1 -11161.019,E2 -11161.019} C_VEL
LIN {X 0,Y 397.323,Z 275.806,A -85,B 0,C 180,E1 -11163.047,E2 -11163.047} C_VEL
LIN {X 0,Y 397.317,Z 275.806,A -85,B 0,C 180,E1 -11166.097,E2 -11166.097} C_VEL
LIN {X 0,Y 397.223,Z 275.819,A -85,B 0,C 180,E1 -11169.167,E2 -11169.167} C_VEL
LIN {X 0,Y 397.208,Z 275.819,A -85,B 0,C 180,E1 -11172.263,E2 -11172.263} C_VEL
LIN {X 0,Y 397.115,Z 275.832,A -85,B 0,C 180,E1 -11175.399,E2 -11175.399} C_VEL
LIN {X 0,Y 397.106,Z 275.833,A -85,B 0,C 180,E1 -11178.58,E2 -11178.58} C_VEL
LIN {X 0,Y 397.088,Z 275.834,A -85,B 0,C 180,E1 -11181.823,E2 -11181.823} C_VEL
LIN {X 0,Y 397.092,Z 275.834,A -85,B 0,C 180,E1 -11185.14,E2 -11185.14} C_VEL
LIN {X 0,Y 397.074,Z 275.835,A -85,B 0,C 180,E1 -11188.551,E2 -11188.551} C_VEL
LIN {X 0,Y 397.078,Z 275.836,A -85,B 0,C 180,E1 -11191.84,E2 -11191.84} C_VEL
LIN {X 0,Y 397.114,Z 275.83,A -85,B 0,C 180,E1 -11194.498,E2 -11194.498} C_VEL
LIN {X 0,Y 397.088,Z 275.833,A -85,B 0,C 180,E1 -11198.281,E2 -11198.281} C_VEL
LIN {X 0,Y 397.051,Z 275.841,A -85,B 0,C 180,E1 -11201.98,E2 -11201.98} C_VEL
LIN {X 0,Y 397.084,Z 275.834,A -85,B 0,C 180,E1 -11205.073,E2 -11205.073} C_VEL
LIN {X 0,Y 397.052,Z 275.84,A -85,B 0,C 180,E1 -11208.027,E2 -11208.027} C_VEL
LIN {X 0,Y 397.093,Z 275.834,A -85,B 0,C 180,E1 -11211.727,E2 -11211.727} C_VEL
LIN {X 0,Y 397.12,Z 275.831,A -85,B 0,C 180,E1 -11215.509,E2 -11215.509} C_VEL
LIN {X 0,Y 397.079,Z 275.834,A -85,B 0,C 180,E1 -11219.12,E2 -11219.12} C_VEL
LIN {X 0,Y 397.063,Z 275.838,A -85,B 0,C 180,E1 -11222.256,E2 -11222.256} C_VEL
LIN {X 0,Y 397.212,Z 275.969,A -85,B 0,C 180,E1 -11224.631,E2 -11224.631} C_VEL
LIN {X 0,Y 398.696,Z 284.712,A -85,B 0,C 180,E1 -11226.85,E2 -11226.85} C_VEL
LIN {X 0,Y 398.656,Z 290.559,A -85,B 0,C 180,E1 -11228.273,E2 -11228.273} C_VEL
LIN {X 0,Y 397.734,Z 303.909,A -85,B 0,C 180,E1 -11231.456,E2 -11231.456} C_VEL
LIN {X 0,Y 396.998,Z 318.285,A -85,B 0,C 180,E1 -11234.856,E2 -11234.856} C_VEL
LIN {X 0,Y 399.454,Z 342.744,A -85,B 0,C 180,E1 -11235.489,E2 -11235.489} C_VEL
LIN {X 0,Y 398.684,Z 397.065,A -85,B 0,C 180,E1 -11236.754,E2 -11236.754} C_VEL
LIN {X 0,Y 398.292,Z 409.661,A -85,B 0,C 180,E1 -11237.26,E2 -11237.26} C_VEL
LIN {X 0,Y 397.895,Z 418.429,A -85,B 0,C 180,E1 -11237.765,E2 -11237.765} C_VEL
LIN {X 0,Y 397.522,Z 427.057,A -85,B 0,C 180,E1 -11238.4,E2 -11238.4} C_VEL
LIN {X 0,Y 397.101,Z 435.383,A -85,B 0,C 180,E1 -11239.163,E2 -11239.163} C_VEL
LIN {X 0,Y 396.832,Z 442.295,A -85,B 0,C 180,E1 -11239.93,E2 -11239.93} C_VEL
LIN {X 0,Y 396.482,Z 450.793,A -85,B 0,C 180,E1 -11241.079,E2 -11241.079} C_VEL
LIN {X 0,Y 396.187,Z 458.335,A -85,B 0,C 180,E1 -11242.356,E2 -11242.356} C_VEL
LIN {X 0,Y 395.964,Z 464.49,A -85,B 0,C 180,E1 -11243.71,E2 -11243.71} C_VEL
LIN {X 0,Y 395.914,Z 468.815,A -85,B 0,C 180,E1 -11244.91,E2 -11244.91} C_VEL
LIN {X 0,Y 395.768,Z 472.949,A -85,B 0,C 180,E1 -11246.438,E2 -11246.438} C_VEL
LIN {X 0,Y 395.868,Z 475.76,A -85,B 0,C 180,E1 -11247.967,E2 -11247.967} C_VEL
LIN {X 0,Y 395.815,Z 476.824,A -85,B 0,C 180,E1 -11248.984,E2 -11248.984} C_VEL
LIN {X 0,Y 395.802,Z 477.367,A -85,B 0,C 180,E1 -11250.002,E2 -11250.002} C_VEL
LIN {X 0,Y 395.799,Z 477.395,A -85,B 0,C 180,E1 -11251.019,E2 -11251.019} C_VEL
LIN {X 0,Y 395.781,Z 476.903,A -85,B 0,C 180,E1 -11252.037,E2 -11252.037} C_VEL
LIN {X 0,Y 395.743,Z 475.814,A -85,B 0,C 180,E1 -11253.056,E2 -11253.056} C_VEL
LIN {X 0,Y 395.882,Z 473.121,A -85,B 0,C 180,E1 -11254.584,E2 -11254.584} C_VEL
LIN {X 0,Y 395.942,Z 469.039,A -85,B 0,C 180,E1 -11256.115,E2 -11256.115} C_VEL
LIN {X 0,Y 396.228,Z 464.547,A -85,B 0,C 180,E1 -11257.39,E2 -11257.39} C_VEL
LIN {X 0,Y 396.575,Z 458.878,A -85,B 0,C 180,E1 -11258.665,E2 -11258.665} C_VEL
LIN {X 0,Y 397.162,Z 451.821,A -85,B 0,C 180,E1 -11259.937,E2 -11259.937} C_VEL
LIN {X 0,Y 397.805,Z 442.758,A -85,B 0,C 180,E1 -11261.208,E2 -11261.208} C_VEL
LIN {X 0,Y 398.302,Z 434.924,A -85,B 0,C 180,E1 -11262.097,E2 -11262.097} C_VEL
LIN {X 0,Y 398.891,Z 426.765,A -85,B 0,C 180,E1 -11262.854,E2 -11262.854} C_VEL
LIN {X 0,Y 399.607,Z 416.588,A -85,B 0,C 180,E1 -11263.607,E2 -11263.607} C_VEL
LIN {X 0,Y 400.352,Z 404.489,A -85,B 0,C 180,E1 -11264.261,E2 -11264.261} C_VEL
LIN {X 0,Y 400.85,Z 394.423,A -85,B 0,C 180,E1 -11264.632,E2 -11264.632} C_VEL
LIN {X 0,Y 402.116,Z 341.325,A -85,B 0,C 180,E1 -11265.97,E2 -11265.97} C_VEL
LIN {X 0,Y 400.482,Z 328.068,A -85,B 0,C 180,E1 -11266.434,E2 -11266.434} C_VEL
LIN {X 0,Y 397.911,Z 314.48,A -85,B 0,C 180,E1 -11267.023,E2 -11267.023} C_VEL
LIN {X 0,Y 398.663,Z 296.856,A -85,B 0,C 180,E1 -11270.647,E2 -11270.647} C_VEL
LIN {X 0,Y 399.149,Z 286.548,A -85,B 0,C 180,E1 -11272.792,E2 -11272.792} C_VEL
LIN {X 0,Y 398.783,Z 282.902,A -85,B 0,C 180,E1 -11273.586,E2 -11273.586} C_VEL
LIN {X 0,Y 397.13,Z 275.833,A -85,B 0,C 180,E1 -11275.262,E2 -11275.262} C_VEL
LIN {X 0,Y 397.074,Z 275.842,A -85,B 0,C 180,E1 -11278.549,E2 -11278.549} C_VEL
LIN {X 0,Y 397.07,Z 275.836,A -85,B 0,C 180,E1 -11281.829,E2 -11281.829} C_VEL
LIN {X 0,Y 397.045,Z 275.84,A -85,B 0,C 180,E1 -11285.484,E2 -11285.484} C_VEL
LIN {X 0,Y 397.1,Z 275.834,A -85,B 0,C 180,E1 -11288.852,E2 -11288.852} C_VEL
LIN {X 0,Y 397.047,Z 275.837,A -85,B 0,C 180,E1 -11292.272,E2 -11292.272} C_VEL
LIN {X 0,Y 397.087,Z 275.836,A -85,B 0,C 180,E1 -11295.07,E2 -11295.07} C_VEL
LIN {X 0,Y 397.062,Z 275.837,A -85,B 0,C 180,E1 -11299.084,E2 -11299.084} C_VEL
LIN {X 0,Y 397.108,Z 275.827,A -85,B 0,C 180,E1 -11301.722,E2 -11301.722} C_VEL
LIN {X 0,Y 397.134,Z 275.826,A -85,B 0,C 180,E1 -11305.504,E2 -11305.504} C_VEL
LIN {X 0,Y 397.094,Z 275.834,A -85,B 0,C 180,E1 -11309.115,E2 -11309.115} C_VEL
LIN {X 0,Y 397.109,Z 275.833,A -85,B 0,C 180,E1 -11312.599,E2 -11312.599} C_VEL
LIN {X 0,Y 397.137,Z 275.832,A -85,B 0,C 180,E1 -11315.978,E2 -11315.978} C_VEL
LIN {X 0,Y 397.155,Z 275.829,A -85,B 0,C 180,E1 -11319.701,E2 -11319.701} C_VEL
LIN {X 0,Y 397.199,Z 276.033,A -85,B 0,C 180,E1 -11320.889,E2 -11320.889} C_VEL
LIN {X 0,Y 399.614,Z 284.946,A -85,B 0,C 180,E1 -11322.599,E2 -11322.599} C_VEL
LIN {X 0,Y 399.679,Z 288.03,A -85,B 0,C 180,E1 -11323.114,E2 -11323.114} C_VEL
LIN {X 0,Y 402.388,Z 302.616,A -85,B 0,C 180,E1 -11323.72,E2 -11323.72} C_VEL
LIN {X 0,Y 402.858,Z 307.594,A -85,B 0,C 180,E1 -11323.888,E2 -11323.888} C_VEL
LIN {X 0,Y 401.084,Z 369.876,A -85,B 0,C 180,E1 -11325.471,E2 -11325.471} C_VEL
LIN {X 0,Y 400.576,Z 381.688,A -85,B 0,C 180,E1 -11325.971,E2 -11325.971} C_VEL
LIN {X 0,Y 400.133,Z 391.054,A -85,B 0,C 180,E1 -11326.538,E2 -11326.538} C_VEL
LIN {X 0,Y 399.688,Z 399.279,A -85,B 0,C 180,E1 -11327.169,E2 -11327.169} C_VEL
LIN {X 0,Y 399.086,Z 407.335,A -85,B 0,C 180,E1 -11327.925,E2 -11327.925} C_VEL
LIN {X 0,Y 398.657,Z 415.063,A -85,B 0,C 180,E1 -11328.814,E2 -11328.814} C_VEL
LIN {X 0,Y 397.938,Z 424.015,A -85,B 0,C 180,E1 -11330.08,E2 -11330.08} C_VEL
LIN {X 0,Y 397.328,Z 430.925,A -85,B 0,C 180,E1 -11331.348,E2 -11331.348} C_VEL
LIN {X 0,Y 397.092,Z 435.455,A -85,B 0,C 180,E1 -11332.368,E2 -11332.368} C_VEL
LIN {X 0,Y 396.713,Z 439.231,A -85,B 0,C 180,E1 -11333.383,E2 -11333.383} C_VEL
LIN {X 0,Y 396.318,Z 442.301,A -85,B 0,C 180,E1 -11334.398,E2 -11334.398} C_VEL
LIN {X 0,Y 396.289,Z 445.618,A -85,B 0,C 180,E1 -11335.927,E2 -11335.927} C_VEL
LIN {X 0,Y 396.096,Z 447.198,A -85,B 0,C 180,E1 -11336.944,E2 -11336.944} C_VEL
LIN {X 0,Y 395.928,Z 448.166,A -85,B 0,C 180,E1 -11337.96,E2 -11337.96} C_VEL
LIN {X 0,Y 395.823,Z 448.571,A -85,B 0,C 180,E1 -11338.978,E2 -11338.978} C_VEL
LIN {X 0,Y 395.803,Z 448.464,A -85,B 0,C 180,E1 -11339.995,E2 -11339.995} C_VEL
LIN {X 0,Y 395.819,Z 447.848,A -85,B 0,C 180,E1 -11341.012,E2 -11341.012} C_VEL
LIN {X 0,Y 395.883,Z 446.711,A -85,B 0,C 180,E1 -11342.03,E2 -11342.03} C_VEL
LIN {X 0,Y 395.962,Z 443.818,A -85,B 0,C 180,E1 -11343.556,E2 -11343.556} C_VEL
LIN {X 0,Y 396.068,Z 439.596,A -85,B 0,C 180,E1 -11345.085,E2 -11345.085} C_VEL
LIN {X 0,Y 396.215,Z 435.058,A -85,B 0,C 180,E1 -11346.326,E2 -11346.326} C_VEL
LIN {X 0,Y 396.539,Z 429.045,A -85,B 0,C 180,E1 -11347.633,E2 -11347.633} C_VEL
LIN {X 0,Y 396.829,Z 421.486,A -85,B 0,C 180,E1 -11348.909,E2 -11348.909} C_VEL
LIN {X 0,Y 397.123,Z 413.999,A -85,B 0,C 180,E1 -11349.93,E2 -11349.93} C_VEL
LIN {X 0,Y 397.569,Z 406.048,A -85,B 0,C 180,E1 -11350.82,E2 -11350.82} C_VEL
LIN {X 0,Y 397.864,Z 397.692,A -85,B 0,C 180,E1 -11351.586,E2 -11351.586} C_VEL
LIN {X 0,Y 398.262,Z 387.169,A -85,B 0,C 180,E1 -11352.349,E2 -11352.349} C_VEL
LIN {X 0,Y 398.609,Z 375.388,A -85,B 0,C 180,E1 -11352.953,E2 -11352.953} C_VEL
LIN {X 0,Y 398.763,Z 365.421,A -85,B 0,C 180,E1 -11353.304,E2 -11353.304} C_VEL
LIN {X 0,Y 399.598,Z 305.637,A -85,B 0,C 180,E1 -11354.684,E2 -11354.684} C_VEL
LIN {X 0,Y 397.182,Z 289.312,A -85,B 0,C 180,E1 -11355.156,E2 -11355.156} C_VEL
LIN {X 0,Y 397.49,Z 279.245,A -85,B 0,C 180,E1 -11358.018,E2 -11358.018} C_VEL
LIN {X 0,Y 397.212,Z 275.819,A -85,B 0,C 180,E1 -11359.033,E2 -11359.033} C_VEL
LIN {X 0,Y 397.083,Z 275.834,A -85,B 0,C 180,E1 -11363.02,E2 -11363.02} C_VEL
LIN {X 0,Y 397.062,Z 275.838,A -85,B 0,C 180,E1 -11366.256,E2 -11366.256} C_VEL
LIN {X 0,Y 397.079,Z 275.836,A -85,B 0,C 180,E1 -11369.856,E2 -11369.856} C_VEL
LIN {X 0,Y 397.097,Z 275.832,A -85,B 0,C 180,E1 -11373.711,E2 -11373.711} C_VEL
LIN {X 0,Y 397.066,Z 275.837,A -85,B 0,C 180,E1 -11377.202,E2 -11377.202} C_VEL
LIN {X 0,Y 397.031,Z 275.842,A -85,B 0,C 180,E1 -11380.432,E2 -11380.432} C_VEL
LIN {X 0,Y 397.069,Z 275.835,A -85,B 0,C 180,E1 -11383.643,E2 -11383.643} C_VEL
LIN {X 0,Y 397.069,Z 275.837,A -85,B 0,C 180,E1 -11386.515,E2 -11386.515} C_VEL
LIN {X 0,Y 397.067,Z 275.838,A -85,B 0,C 180,E1 -11390.416,E2 -11390.416} C_VEL
LIN {X 0,Y 397.069,Z 275.836,A -85,B 0,C 180,E1 -11394.26,E2 -11394.26} C_VEL
LIN {X 0,Y 397.073,Z 275.837,A -85,B 0,C 180,E1 -11396.722,E2 -11396.722} C_VEL
LIN {X 0,Y 397.08,Z 275.834,A -85,B 0,C 180,E1 -11400.291,E2 -11400.291} C_VEL
LIN {X 0,Y 397.149,Z 275.826,A -85,B 0,C 180,E1 -11402.605,E2 -11402.605} C_VEL
LIN {X 0,Y 397.085,Z 275.834,A -85,B 0,C 180,E1 -11405.977,E2 -11405.977} C_VEL
LIN {X 0,Y 397.089,Z 275.836,A -85,B 0,C 180,E1 -11409.701,E2 -11409.701} C_VEL
LIN {X 0,Y 397.131,Z 275.828,A -85,B 0,C 180,E1 -11412.841,E2 -11412.841} C_VEL
LIN {X 0,Y 397.176,Z 275.822,A -85,B 0,C 180,E1 -11416.699,E2 -11416.699} C_VEL
LIN {X 0,Y 397.175,Z 275.824,A -85,B 0,C 180,E1 -11419.806,E2 -11419.806} C_VEL
LIN {X 0,Y 397.301,Z 275.807,A -85,B 0,C 180,E1 -11422.885,E2 -11422.885} C_VEL
LIN {X 0,Y 397.207,Z 275.818,A -85,B 0,C 180,E1 -11424.923,E2 -11424.923} C_VEL
LIN {X 0,Y 397.396,Z 275.796,A -85,B 0,C 180,E1 -11427.971,E2 -11427.971} C_VEL
LIN {X 0,Y 397.525,Z 275.78,A -85,B 0,C 180,E1 -11429.998,E2 -11429.998} C_VEL
LIN {X 0,Y 397.332,Z 275.803,A -85,B 0,C 180,E1 -11433.04,E2 -11433.04} C_VEL
LIN {X 0,Y 397.318,Z 275.806,A -85,B 0,C 180,E1 -11436.091,E2 -11436.091} C_VEL
LIN {X 0,Y 397.198,Z 275.819,A -85,B 0,C 180,E1 -11439.188,E2 -11439.188} C_VEL
LIN {X 0,Y 397.173,Z 275.824,A -85,B 0,C 180,E1 -11442.258,E2 -11442.258} C_VEL
LIN {X 0,Y 397.143,Z 275.825,A -85,B 0,C 180,E1 -11443.604,E2 -11443.604} C_VEL
LIN {X 0,Y 396.445,Z 275.916,A -85,B 0,C 180,E1 -11444.45,E2 -11444.45} C_VEL
LIN {X 0,Y 393.596,Z 276.269,A -85,B 0,C 180,E1 -11445.825,E2 -11445.825} C_VEL
LIN {X 0,Y 391.193,Z 276.569,A -85,B 0,C 180,E1 -11446.937,E2 -11446.937} C_VEL
LIN {X 0,Y 390.147,Z 276.698,A -85,B 0,C 180,E1 -11447.795,E2 -11447.795} C_VEL
LIN {X 0,Y 390.052,Z 276.709,A -85,B 0,C 180,E1 -11448.086,E2 -11448.086} C_VEL
LIN {X 0,Y 389.998,Z 276.718,A -85,B 0,C 180,E1 -11451.123,E2 -11451.123} C_VEL
LIN {X 0,Y 390.024,Z 276.715,A -85,B 0,C 180,E1 -11454.482,E2 -11454.482} C_VEL
LIN {X 0,Y 390.061,Z 276.709,A -85,B 0,C 180,E1 -11458.027,E2 -11458.027} C_VEL
LIN {X 0,Y 389.972,Z 276.72,A -85,B 0,C 180,E1 -11461.506,E2 -11461.506} C_VEL
LIN {X 0,Y 390.032,Z 276.715,A -85,B 0,C 180,E1 -11465.21,E2 -11465.21} C_VEL
LIN {X 0,Y 390.045,Z 276.712,A -85,B 0,C 180,E1 -11469.095,E2 -11469.095} C_VEL
LIN {X 0,Y 390.073,Z 276.707,A -85,B 0,C 180,E1 -11472.39,E2 -11472.39} C_VEL
LIN {X 0,Y 390.071,Z 276.709,A -85,B 0,C 180,E1 -11475.369,E2 -11475.369} C_VEL
LIN {X 0,Y 390.059,Z 276.708,A -85,B 0,C 180,E1 -11478.2,E2 -11478.2} C_VEL
LIN {X 0,Y 390.051,Z 276.711,A -85,B 0,C 180,E1 -11480.912,E2 -11480.912} C_VEL
LIN {X 0,Y 390.044,Z 276.711,A -85,B 0,C 180,E1 -11484.798,E2 -11484.798} C_VEL
LIN {X 0,Y 389.984,Z 276.718,A -85,B 0,C 180,E1 -11488.5,E2 -11488.5} C_VEL
LIN {X 0,Y 390.081,Z 276.709,A -85,B 0,C 180,E1 -11492.075,E2 -11492.075} C_VEL
LIN {X 0,Y 390.04,Z 276.713,A -85,B 0,C 180,E1 -11495.524,E2 -11495.524} C_VEL
LIN {X 0,Y 390.056,Z 276.711,A -85,B 0,C 180,E1 -11499.535,E2 -11499.535} C_VEL
LIN {X 0,Y 390.109,Z 276.702,A -85,B 0,C 180,E1 -11503.253,E2 -11503.253} C_VEL
LIN {X 0,Y 390.169,Z 276.697,A -85,B 0,C 180,E1 -11506.567,E2 -11506.567} C_VEL
LIN {X 0,Y 390.142,Z 276.699,A -85,B 0,C 180,E1 -11509.628,E2 -11509.628} C_VEL
LIN {X 0,Y 390.257,Z 276.686,A -85,B 0,C 180,E1 -11512.764,E2 -11512.764} C_VEL
LIN {X 0,Y 390.193,Z 276.694,A -85,B 0,C 180,E1 -11514.839,E2 -11514.839} C_VEL
LIN {X 0,Y 390.39,Z 276.669,A -85,B 0,C 180,E1 -11517.942,E2 -11517.942} C_VEL
LIN {X 0,Y 390.275,Z 276.683,A -85,B 0,C 180,E1 -11521.037,E2 -11521.037} C_VEL
LIN {X 0,Y 390.26,Z 276.685,A -85,B 0,C 180,E1 -11523.102,E2 -11523.102} C_VEL
LIN {X 0,Y 390.271,Z 276.684,A -85,B 0,C 180,E1 -11526.208,E2 -11526.208} C_VEL
LIN {X 0,Y 390.18,Z 276.695,A -85,B 0,C 180,E1 -11529.334,E2 -11529.334} C_VEL
LIN {X 0,Y 390.16,Z 276.698,A -85,B 0,C 180,E1 -11532.488,E2 -11532.488} C_VEL
LIN {X 0,Y 390.058,Z 276.709,A -85,B 0,C 180,E1 -11535.685,E2 -11535.685} C_VEL
LIN {X 0,Y 390.068,Z 276.709,A -85,B 0,C 180,E1 -11538.928,E2 -11538.928} C_VEL
LIN {X 0,Y 390.028,Z 276.712,A -85,B 0,C 180,E1 -11542.239,E2 -11542.239} C_VEL
LIN {X 0,Y 390.045,Z 276.712,A -85,B 0,C 180,E1 -11545.726,E2 -11545.726} C_VEL
LIN {X 0,Y 390.029,Z 276.714,A -85,B 0,C 180,E1 -11549.116,E2 -11549.116} C_VEL
LIN {X 0,Y 390.039,Z 276.712,A -85,B 0,C 180,E1 -11552.726,E2 -11552.726} C_VEL
LIN {X 0,Y 390.04,Z 276.714,A -85,B 0,C 180,E1 -11555.826,E2 -11555.826} C_VEL
LIN {X 0,Y 390.035,Z 276.713,A -85,B 0,C 180,E1 -11559.216,E2 -11559.216} C_VEL
LIN {X 0,Y 390.03,Z 276.713,A -85,B 0,C 180,E1 -11562.376,E2 -11562.376} C_VEL
LIN {X 0,Y 390.04,Z 276.713,A -85,B 0,C 180,E1 -11565.357,E2 -11565.357} C_VEL
LIN {X 0,Y 390.015,Z 276.717,A -85,B 0,C 180,E1 -11568.188,E2 -11568.188} C_VEL
LIN {X 0,Y 390.06,Z 276.708,A -85,B 0,C 180,E1 -11570.907,E2 -11570.907} C_VEL
LIN {X 0,Y 390.072,Z 276.707,A -85,B 0,C 180,E1 -11574.795,E2 -11574.795} C_VEL
LIN {X 0,Y 390.025,Z 276.716,A -85,B 0,C 180,E1 -11578.498,E2 -11578.498} C_VEL
LIN {X 0,Y 390.022,Z 276.715,A -85,B 0,C 180,E1 -11582.006,E2 -11582.006} C_VEL
LIN {X 0,Y 390.155,Z 276.883,A -85,B 0,C 180,E1 -11584.53,E2 -11584.53} C_VEL
LIN {X 0,Y 391.78,Z 286.615,A -85,B 0,C 180,E1 -11587.037,E2 -11587.037} C_VEL
LIN {X 0,Y 391.332,Z 295.311,A -85,B 0,C 180,E1 -11589.17,E2 -11589.17} C_VEL
LIN {X 0,Y 390.345,Z 310.763,A -85,B 0,C 180,E1 -11592.919,E2 -11592.919} C_VEL
LIN {X 0,Y 389.961,Z 318.015,A -85,B 0,C 180,E1 -11594.668,E2 -11594.668} C_VEL
LIN {X 0,Y 392.456,Z 342.647,A -85,B 0,C 180,E1 -11595.333,E2 -11595.333} C_VEL
LIN {X 0,Y 391.638,Z 396.15,A -85,B 0,C 180,E1 -11596.61,E2 -11596.61} C_VEL
LIN {X 0,Y 391.268,Z 408.442,A -85,B 0,C 180,E1 -11597.093,E2 -11597.093} C_VEL
LIN {X 0,Y 390.835,Z 418.336,A -85,B 0,C 180,E1 -11597.672,E2 -11597.672} C_VEL
LIN {X 0,Y 390.456,Z 426.928,A -85,B 0,C 180,E1 -11598.319,E2 -11598.319} C_VEL
LIN {X 0,Y 390.026,Z 435.231,A -85,B 0,C 180,E1 -11599.096,E2 -11599.096} C_VEL
LIN {X 0,Y 389.752,Z 442.128,A -85,B 0,C 180,E1 -11599.876,E2 -11599.876} C_VEL
LIN {X 0,Y 389.479,Z 447.991,A -85,B 0,C 180,E1 -11600.656,E2 -11600.656} C_VEL
LIN {X 0,Y 389.231,Z 454.543,A -85,B 0,C 180,E1 -11601.697,E2 -11601.697} C_VEL
LIN {X 0,Y 389.043,Z 459.976,A -85,B 0,C 180,E1 -11602.737,E2 -11602.737} C_VEL
LIN {X 0,Y 388.885,Z 464.482,A -85,B 0,C 180,E1 -11603.777,E2 -11603.777} C_VEL
LIN {X 0,Y 388.825,Z 468.209,A -85,B 0,C 180,E1 -11604.817,E2 -11604.817} C_VEL
LIN {X 0,Y 388.745,Z 471.238,A -85,B 0,C 180,E1 -11605.855,E2 -11605.855} C_VEL
LIN {X 0,Y 388.687,Z 473.606,A -85,B 0,C 180,E1 -11606.892,E2 -11606.892} C_VEL
LIN {X 0,Y 388.781,Z 475.318,A -85,B 0,C 180,E1 -11607.93,E2 -11607.93} C_VEL
LIN {X 0,Y 388.747,Z 476.451,A -85,B 0,C 180,E1 -11608.966,E2 -11608.966} C_VEL
LIN {X 0,Y 388.731,Z 477.057,A -85,B 0,C 180,E1 -11610.002,E2 -11610.002} C_VEL
LIN {X 0,Y 388.729,Z 477.146,A -85,B 0,C 180,E1 -11611.038,E2 -11611.038} C_VEL
LIN {X 0,Y 388.679,Z 476.697,A -85,B 0,C 180,E1 -11612.074,E2 -11612.074} C_VEL
LIN {X 0,Y 388.651,Z 475.628,A -85,B 0,C 180,E1 -11613.111,E2 -11613.111} C_VEL
LIN {X 0,Y 388.815,Z 473.061,A -85,B 0,C 180,E1 -11614.667,E2 -11614.667} C_VEL
LIN {X 0,Y 388.886,Z 468.905,A -85,B 0,C 180,E1 -11616.279,E2 -11616.279} C_VEL
LIN {X 0,Y 389.246,Z 463.625,A -85,B 0,C 180,E1 -11617.784,E2 -11617.784} C_VEL
LIN {X 0,Y 389.637,Z 457.798,A -85,B 0,C 180,E1 -11619.082,E2 -11619.082} C_VEL
LIN {X 0,Y 390.268,Z 450.483,A -85,B 0,C 180,E1 -11620.376,E2 -11620.376} C_VEL
LIN {X 0,Y 390.955,Z 442.178,A -85,B 0,C 180,E1 -11621.538,E2 -11621.538} C_VEL
LIN {X 0,Y 391.446,Z 434.361,A -85,B 0,C 180,E1 -11622.443,E2 -11622.443} C_VEL
LIN {X 0,Y 392.145,Z 426.21,A -85,B 0,C 180,E1 -11623.211,E2 -11623.211} C_VEL
LIN {X 0,Y 392.922,Z 416.068,A -85,B 0,C 180,E1 -11623.975,E2 -11623.975} C_VEL
LIN {X 0,Y 393.681,Z 403.865,A -85,B 0,C 180,E1 -11624.64,E2 -11624.64} C_VEL
LIN {X 0,Y 394.235,Z 393.709,A -85,B 0,C 180,E1 -11625.015,E2 -11625.015} C_VEL
LIN {X 0,Y 395.619,Z 342.303,A -85,B 0,C 180,E1 -11626.348,E2 -11626.348} C_VEL
LIN {X 0,Y 394.093,Z 329.671,A -85,B 0,C 180,E1 -11626.816,E2 -11626.816} C_VEL
LIN {X 0,Y 391.104,Z 314.076,A -85,B 0,C 180,E1 -11627.507,E2 -11627.507} C_VEL
LIN {X 0,Y 391.984,Z 296.57,A -85,B 0,C 180,E1 -11631.194,E2 -11631.194} C_VEL
LIN {X 0,Y 392.32,Z 287.055,A -85,B 0,C 180,E1 -11633.212,E2 -11633.212} C_VEL
LIN {X 0,Y 390.428,Z 278.162,A -85,B 0,C 180,E1 -11635.312,E2 -11635.312} C_VEL
LIN {X 0,Y 390.06,Z 276.714,A -85,B 0,C 180,E1 -11635.72,E2 -11635.72} C_VEL
LIN {X 0,Y 390.033,Z 276.719,A -85,B 0,C 180,E1 -11639.113,E2 -11639.113} C_VEL
LIN {X 0,Y 390.011,Z 276.719,A -85,B 0,C 180,E1 -11642.726,E2 -11642.726} C_VEL
LIN {X 0,Y 390.022,Z 276.714,A -85,B 0,C 180,E1 -11646.489,E2 -11646.489} C_VEL
LIN {X 0,Y 390.043,Z 276.712,A -85,B 0,C 180,E1 -11649.209,E2 -11649.209} C_VEL
LIN {X 0,Y 390.024,Z 276.712,A -85,B 0,C 180,E1 -11652.367,E2 -11652.367} C_VEL
LIN {X 0,Y 390.021,Z 276.713,A -85,B 0,C 180,E1 -11655.347,E2 -11655.347} C_VEL
LIN {X 0,Y 390.021,Z 276.71,A -85,B 0,C 180,E1 -11658.181,E2 -11658.181} C_VEL
LIN {X 0,Y 390.075,Z 276.708,A -85,B 0,C 180,E1 -11660.902,E2 -11660.902} C_VEL
LIN {X 0,Y 390.086,Z 276.707,A -85,B 0,C 180,E1 -11664.789,E2 -11664.789} C_VEL
LIN {X 0,Y 390.04,Z 276.713,A -85,B 0,C 180,E1 -11668.493,E2 -11668.493} C_VEL
LIN {X 0,Y 390.046,Z 276.712,A -85,B 0,C 180,E1 -11672.06,E2 -11672.06} C_VEL
LIN {X 0,Y 390.069,Z 276.715,A -85,B 0,C 180,E1 -11675.514,E2 -11675.514} C_VEL
LIN {X 0,Y 390.071,Z 276.712,A -85,B 0,C 180,E1 -11678.874,E2 -11678.874} C_VEL
LIN {X 0,Y 390.128,Z 276.755,A -85,B 0,C 180,E1 -11680.357,E2 -11680.357} C_VEL
LIN {X 0,Y 392.816,Z 286.474,A -85,B 0,C 180,E1 -11682.288,E2 -11682.288} C_VEL
LIN {X 0,Y 393.098,Z 288.543,A -85,B 0,C 180,E1 -11682.648,E2 -11682.648} C_VEL
LIN {X 0,Y 395.972,Z 303.499,A -85,B 0,C 180,E1 -11683.297,E2 -11683.297} C_VEL
LIN {X 0,Y 396.44,Z 307.834,A -85,B 0,C 180,E1 -11683.458,E2 -11683.458} C_VEL
LIN {X 0,Y 394.463,Z 370.747,A -85,B 0,C 180,E1 -11685.123,E2 -11685.123} C_VEL
LIN {X 0,Y 393.896,Z 382.853,A -85,B 0,C 180,E1 -11685.662,E2 -11685.662} C_VEL
LIN {X 0,Y 393.372,Z 392.929,A -85,B 0,C 180,E1 -11686.302,E2 -11686.302} C_VEL
LIN {X 0,Y 392.781,Z 402.33,A -85,B 0,C 180,E1 -11687.071,E2 -11687.071} C_VEL
LIN {X 0,Y 392.116,Z 412.169,A -85,B 0,C 180,E1 -11688.1,E2 -11688.1} C_VEL
LIN {X 0,Y 391.475,Z 419.923,A -85,B 0,C 180,E1 -11689.13,E2 -11689.13} C_VEL
LIN {X 0,Y 390.881,Z 426.331,A -85,B 0,C 180,E1 -11690.16,E2 -11690.16} C_VEL
LIN {X 0,Y 390.267,Z 432.866,A -85,B 0,C 180,E1 -11691.451,E2 -11691.451} C_VEL
LIN {X 0,Y 389.923,Z 438.078,A -85,B 0,C 180,E1 -11692.747,E2 -11692.747} C_VEL
LIN {X 0,Y 389.279,Z 442.868,A -85,B 0,C 180,E1 -11694.296,E2 -11694.296} C_VEL
LIN {X 0,Y 389.226,Z 446.088,A -85,B 0,C 180,E1 -11695.853,E2 -11695.853} C_VEL
LIN {X 0,Y 389.044,Z 447.608,A -85,B 0,C 180,E1 -11696.888,E2 -11696.888} C_VEL
LIN {X 0,Y 388.866,Z 448.554,A -85,B 0,C 180,E1 -11697.923,E2 -11697.923} C_VEL
LIN {X 0,Y 388.754,Z 448.891,A -85,B 0,C 180,E1 -11698.959,E2 -11698.959} C_VEL
LIN {X 0,Y 388.732,Z 448.71,A -85,B 0,C 180,E1 -11699.995,E2 -11699.995} C_VEL
LIN {X 0,Y 388.75,Z 448.021,A -85,B 0,C 180,E1 -11701.031,E2 -11701.031} C_VEL
LIN {X 0,Y 388.785,Z 446.818,A -85,B 0,C 180,E1 -11702.067,E2 -11702.067} C_VEL
LIN {X 0,Y 388.867,Z 443.846,A -85,B 0,C 180,E1 -11703.621,E2 -11703.621} C_VEL
LIN {X 0,Y 388.99,Z 439.536,A -85,B 0,C 180,E1 -11705.177,E2 -11705.177} C_VEL
LIN {X 0,Y 389.257,Z 433.551,A -85,B 0,C 180,E1 -11706.765,E2 -11706.765} C_VEL
LIN {X 0,Y 389.507,Z 427.26,A -85,B 0,C 180,E1 -11708.033,E2 -11708.033} C_VEL
LIN {X 0,Y 389.778,Z 420.968,A -85,B 0,C 180,E1 -11709.072,E2 -11709.072} C_VEL
LIN {X 0,Y 390.118,Z 413.325,A -85,B 0,C 180,E1 -11710.11,E2 -11710.11} C_VEL
LIN {X 0,Y 390.572,Z 405.181,A -85,B 0,C 180,E1 -11711.016,E2 -11711.016} C_VEL
LIN {X 0,Y 390.966,Z 395.016,A -85,B 0,C 180,E1 -11711.924,E2 -11711.924} C_VEL
LIN {X 0,Y 391.366,Z 384.261,A -85,B 0,C 180,E1 -11712.636,E2 -11712.636} C_VEL
LIN {X 0,Y 391.614,Z 374.417,A -85,B 0,C 180,E1 -11713.122,E2 -11713.122} C_VEL
LIN {X 0,Y 391.761,Z 363.942,A -85,B 0,C 180,E1 -11713.48,E2 -11713.48} C_VEL
LIN {X 0,Y 392.604,Z 306.405,A -85,B 0,C 180,E1 -11714.835,E2 -11714.835} C_VEL
LIN {X 0,Y 390.133,Z 289.553,A -85,B 0,C 180,E1 -11715.336,E2 -11715.336} C_VEL
LIN {X 0,Y 390.44,Z 280.937,A -85,B 0,C 180,E1 -11717.812,E2 -11717.812} C_VEL
LIN {X 0,Y 390.176,Z 276.695,A -85,B 0,C 180,E1 -11719.117,E2 -11719.117} C_VEL
LIN {X 0,Y 390.046,Z 276.71,A -85,B 0,C 180,E1 -11723.347,E2 -11723.347} C_VEL
LIN {X 0,Y 390.015,Z 276.716,A -85,B 0,C 180,E1 -11726.768,E2 -11726.768} C_VEL
LIN {X 0,Y 390.018,Z 276.716,A -85,B 0,C 180,E1 -11730.294,E2 -11730.294} C_VEL
LIN {X 0,Y 390.048,Z 276.712,A -85,B 0,C 180,E1 -11734.018,E2 -11734.018} C_VEL
LIN {X 0,Y 390.015,Z 276.714,A -85,B 0,C 180,E1 -11737.543,E2 -11737.543} C_VEL
LIN {X 0,Y 389.994,Z 276.719,A -85,B 0,C 180,E1 -11740.809,E2 -11740.809} C_VEL
LIN {X 0,Y 390.023,Z 276.713,A -85,B 0,C 180,E1 -11743.88,E2 -11743.88} C_VEL
LIN {X 0,Y 390.024,Z 276.715,A -85,B 0,C 180,E1 -11746.783,E2 -11746.783} C_VEL
LIN {X 0,Y 390.021,Z 276.714,A -85,B 0,C 180,E1 -11749.555,E2 -11749.555} C_VEL
LIN {X 0,Y 390.004,Z 276.717,A -85,B 0,C 180,E1 -11752.444,E2 -11752.444} C_VEL
LIN {X 0,Y 390.029,Z 276.712,A -85,B 0,C 180,E1 -11755.97,E2 -11755.97} C_VEL
LIN {X 0,Y 390.003,Z 276.716,A -85,B 0,C 180,E1 -11759.864,E2 -11759.864} C_VEL
LIN {X 0,Y 390.068,Z 276.709,A -85,B 0,C 180,E1 -11763.227,E2 -11763.227} C_VEL
LIN {X 0,Y 390.059,Z 276.71,A -85,B 0,C 180,E1 -11766.746,E2 -11766.746} C_VEL
LIN {X 0,Y 390.054,Z 276.711,A -85,B 0,C 180,E1 -11769.979,E2 -11769.979} C_VEL
LIN {X 0,Y 390.086,Z 276.707,A -85,B 0,C 180,E1 -11773.244,E2 -11773.244} C_VEL
LIN {X 0,Y 390.142,Z 276.698,A -85,B 0,C 180,E1 -11776.558,E2 -11776.558} C_VEL
LIN {X 0,Y 390.125,Z 276.702,A -85,B 0,C 180,E1 -11779.62,E2 -11779.62} C_VEL
LIN {X 0,Y 390.252,Z 276.684,A -85,B 0,C 180,E1 -11782.756,E2 -11782.756} C_VEL
LIN {X 0,Y 390.178,Z 276.693,A -85,B 0,C 180,E1 -11784.831,E2 -11784.831} C_VEL
LIN {X 0,Y 390.365,Z 276.672,A -85,B 0,C 180,E1 -11787.935,E2 -11787.935} C_VEL
LIN {X 0,Y 390.495,Z 276.656,A -85,B 0,C 180,E1 -11789.998,E2 -11789.998} C_VEL
LIN {X 0,Y 390.291,Z 276.679,A -85,B 0,C 180,E1 -11793.095,E2 -11793.095} C_VEL
LIN {X 0,Y 390.272,Z 276.684,A -85,B 0,C 180,E1 -11796.201,E2 -11796.201} C_VEL
LIN {X 0,Y 390.153,Z 276.697,A -85,B 0,C 180,E1 -11799.328,E2 -11799.328} C_VEL
LIN {X 0,Y 390.121,Z 276.703,A -85,B 0,C 180,E1 -11802.483,E2 -11802.483} C_VEL
LIN {X 0,Y 390.081,Z 276.706,A -85,B 0,C 180,E1 -11805.677,E2 -11805.677} C_VEL
LIN {X 0,Y 390.052,Z 276.709,A -85,B 0,C 180,E1 -11808.086,E2 -11808.086} C_VEL
LIN {X 0,Y 389.343,Z 276.8,A -85,B 0,C 180,E1 -11808.948,E2 -11808.948} C_VEL
LIN {X 0,Y 386.43,Z 277.163,A -85,B 0,C 180,E1 -11810.348,E2 -11810.348} C_VEL
LIN {X 0,Y 384.01,Z 277.462,A -85,B 0,C 180,E1 -11811.479,E2 -11811.479} C_VEL
LIN {X 0,Y 383.011,Z 277.589,A -85,B 0,C 180,E1 -11812.355,E2 -11812.355} C_VEL
LIN {X 0,Y 382.95,Z 277.596,A -85,B 0,C 180,E1 -11812.651,E2 -11812.651} C_VEL
LIN {X 0,Y 383.024,Z 277.586,A -85,B 0,C 180,E1 -11816.125,E2 -11816.125} C_VEL
LIN {X 0,Y 382.994,Z 277.591,A -85,B 0,C 180,E1 -11818.494,E2 -11818.494} C_VEL
LIN {X 0,Y 382.956,Z 277.593,A -85,B 0,C 180,E1 -11822.152,E2 -11822.152} C_VEL
LIN {X 0,Y 382.965,Z 277.594,A -85,B 0,C 180,E1 -11824.671,E2 -11824.671} C_VEL
LIN {X 0,Y 382.952,Z 277.593,A -85,B 0,C 180,E1 -11827.907,E2 -11827.907} C_VEL
LIN {X 0,Y 382.997,Z 277.591,A -85,B 0,C 180,E1 -11831.343,E2 -11831.343} C_VEL
LIN {X 0,Y 383.023,Z 277.585,A -85,B 0,C 180,E1 -11834.318,E2 -11834.318} C_VEL
LIN {X 0,Y 383.03,Z 277.586,A -85,B 0,C 180,E1 -11837.253,E2 -11837.253} C_VEL
LIN {X 0,Y 382.978,Z 277.59,A -85,B 0,C 180,E1 -11840.416,E2 -11840.416} C_VEL
LIN {X 0,Y 382.985,Z 277.591,A -85,B 0,C 180,E1 -11844.049,E2 -11844.049} C_VEL
LIN {X 0,Y 382.947,Z 277.597,A -85,B 0,C 180,E1 -11847.583,E2 -11847.583} C_VEL
LIN {X 0,Y 382.954,Z 277.594,A -85,B 0,C 180,E1 -11850.305,E2 -11850.305} C_VEL
LIN {X 0,Y 383.044,Z 277.586,A -85,B 0,C 180,E1 -11854.026,E2 -11854.026} C_VEL
LIN {X 0,Y 382.958,Z 277.594,A -85,B 0,C 180,E1 -11857.339,E2 -11857.339} C_VEL
LIN {X 0,Y 383.028,Z 277.584,A -85,B 0,C 180,E1 -11860.721,E2 -11860.721} C_VEL
LIN {X 0,Y 383.052,Z 277.584,A -85,B 0,C 180,E1 -11864.032,E2 -11864.032} C_VEL
LIN {X 0,Y 383.11,Z 277.574,A -85,B 0,C 180,E1 -11867.289,E2 -11867.289} C_VEL
LIN {X 0,Y 383.119,Z 277.577,A -85,B 0,C 180,E1 -11870.503,E2 -11870.503} C_VEL
LIN {X 0,Y 383.247,Z 277.558,A -85,B 0,C 180,E1 -11873.689,E2 -11873.689} C_VEL
LIN {X 0,Y 383.356,Z 277.545,A -85,B 0,C 180,E1 -11877.904,E2 -11877.904} C_VEL
LIN {X 0,Y 383.364,Z 277.544,A -85,B 0,C 180,E1 -11882.106,E2 -11882.106} C_VEL
LIN {X 0,Y 383.227,Z 277.562,A -85,B 0,C 180,E1 -11886.322,E2 -11886.322} C_VEL
LIN {X 0,Y 383.131,Z 277.572,A -85,B 0,C 180,E1 -11889.507,E2 -11889.507} C_VEL
LIN {X 0,Y 383.116,Z 277.574,A -85,B 0,C 180,E1 -11893.541,E2 -11893.541} C_VEL
LIN {X 0,Y 383.045,Z 277.584,A -85,B 0,C 180,E1 -11897.439,E2 -11897.439} C_VEL
LIN {X 0,Y 383.022,Z 277.587,A -85,B 0,C 180,E1 -11900.651,E2 -11900.651} C_VEL
LIN {X 0,Y 383.003,Z 277.588,A -85,B 0,C 180,E1 -11903.814,E2 -11903.814} C_VEL
LIN {X 0,Y 382.987,Z 277.592,A -85,B 0,C 180,E1 -11907.312,E2 -11907.312} C_VEL
LIN {X 0,Y 382.979,Z 277.592,A -85,B 0,C 180,E1 -11910.923,E2 -11910.923} C_VEL
LIN {X 0,Y 383.009,Z 277.586,A -85,B 0,C 180,E1 -11914.673,E2 -11914.673} C_VEL
LIN {X 0,Y 382.991,Z 277.592,A -85,B 0,C 180,E1 -11917.906,E2 -11917.906} C_VEL
LIN {X 0,Y 382.961,Z 277.595,A -85,B 0,C 180,E1 -11921.355,E2 -11921.355} C_VEL
LIN {X 0,Y 382.989,Z 277.59,A -85,B 0,C 180,E1 -11924.306,E2 -11924.306} C_VEL
LIN {X 0,Y 382.983,Z 277.591,A -85,B 0,C 180,E1 -11927.24,E2 -11927.24} C_VEL
LIN {X 0,Y 382.988,Z 277.591,A -85,B 0,C 180,E1 -11930.423,E2 -11930.423} C_VEL
LIN {X 0,Y 383.017,Z 277.588,A -85,B 0,C 180,E1 -11934.046,E2 -11934.046} C_VEL
LIN {X 0,Y 382.989,Z 277.59,A -85,B 0,C 180,E1 -11937.582,E2 -11937.582} C_VEL
LIN {X 0,Y 382.979,Z 277.593,A -85,B 0,C 180,E1 -11940.302,E2 -11940.302} C_VEL
LIN {X 0,Y 383.089,Z 277.616,A -85,B 0,C 180,E1 -11944.386,E2 -11944.386} C_VEL
LIN {X 0,Y 384.698,Z 287.083,A -85,B 0,C 180,E1 -11946.875,E2 -11946.875} C_VEL
LIN {X 0,Y 384.364,Z 294.925,A -85,B 0,C 180,E1 -11948.838,E2 -11948.838} C_VEL
LIN {X 0,Y 383.451,Z 308.571,A -85,B 0,C 180,E1 -11952.214,E2 -11952.214} C_VEL
LIN {X 0,Y 382.911,Z 317.727,A -85,B 0,C 180,E1 -11954.466,E2 -11954.466} C_VEL
LIN {X 0,Y 385.443,Z 342.76,A -85,B 0,C 180,E1 -11955.179,E2 -11955.179} C_VEL
LIN {X 0,Y 384.602,Z 396.348,A -85,B 0,C 180,E1 -11956.495,E2 -11956.495} C_VEL
LIN {X 0,Y 384.231,Z 408.419,A -85,B 0,C 180,E1 -11956.987,E2 -11956.987} C_VEL
LIN {X 0,Y 383.777,Z 418.24,A -85,B 0,C 180,E1 -11957.576,E2 -11957.576} C_VEL
LIN {X 0,Y 383.39,Z 426.799,A -85,B 0,C 180,E1 -11958.235,E2 -11958.235} C_VEL
LIN {X 0,Y 382.953,Z 435.082,A -85,B 0,C 180,E1 -11959.026,E2 -11959.026} C_VEL
LIN {X 0,Y 382.673,Z 441.965,A -85,B 0,C 180,E1 -11959.82,E2 -11959.82} C_VEL
LIN {X 0,Y 382.359,Z 448.693,A -85,B 0,C 180,E1 -11960.747,E2 -11960.747} C_VEL
LIN {X 0,Y 382.105,Z 455.094,A -85,B 0,C 180,E1 -11961.807,E2 -11961.807} C_VEL
LIN {X 0,Y 381.95,Z 460.397,A -85,B 0,C 180,E1 -11962.867,E2 -11962.867} C_VEL
LIN {X 0,Y 381.812,Z 464.027,A -85,B 0,C 180,E1 -11963.727,E2 -11963.727} C_VEL
LIN {X 0,Y 381.75,Z 469.172,A -85,B 0,C 180,E1 -11965.25,E2 -11965.25} C_VEL
LIN {X 0,Y 381.609,Z 471.892,A -85,B 0,C 180,E1 -11966.306,E2 -11966.306} C_VEL
LIN {X 0,Y 381.696,Z 474.851,A -85,B 0,C 180,E1 -11967.891,E2 -11967.891} C_VEL
LIN {X 0,Y 381.68,Z 476.059,A -85,B 0,C 180,E1 -11968.947,E2 -11968.947} C_VEL
LIN {X 0,Y 381.662,Z 476.738,A -85,B 0,C 180,E1 -11970.002,E2 -11970.002} C_VEL
LIN {X 0,Y 381.643,Z 476.901,A -85,B 0,C 180,E1 -11971.057,E2 -11971.057} C_VEL
LIN {X 0,Y 381.578,Z 476.479,A -85,B 0,C 180,E1 -11972.113,E2 -11972.113} C_VEL
LIN {X 0,Y 381.564,Z 475.451,A -85,B 0,C 180,E1 -11973.169,E2 -11973.169} C_VEL
LIN {X 0,Y 381.728,Z 472.986,A -85,B 0,C 180,E1 -11974.754,E2 -11974.754} C_VEL
LIN {X 0,Y 381.822,Z 469.097,A -85,B 0,C 180,E1 -11976.342,E2 -11976.342} C_VEL
LIN {X 0,Y 382.145,Z 464.732,A -85,B 0,C 180,E1 -11977.664,E2 -11977.664} C_VEL
LIN {X 0,Y 382.54,Z 459.238,A -85,B 0,C 180,E1 -11978.986,E2 -11978.986} C_VEL
LIN {X 0,Y 383.05,Z 453.877,A -85,B 0,C 180,E1 -11980.04,E2 -11980.04} C_VEL
LIN {X 0,Y 383.641,Z 447.455,A -85,B 0,C 180,E1 -11981.092,E2 -11981.092} C_VEL
LIN {X 0,Y 384.276,Z 439.695,A -85,B 0,C 180,E1 -11982.143,E2 -11982.143} C_VEL
LIN {X 0,Y 385.125,Z 430.142,A -85,B 0,C 180,E1 -11983.187,E2 -11983.187} C_VEL
LIN {X 0,Y 385.84,Z 420.991,A -85,B 0,C 180,E1 -11983.968,E2 -11983.968} C_VEL
LIN {X 0,Y 386.593,Z 410.161,A -85,B 0,C 180,E1 -11984.679,E2 -11984.679} C_VEL
LIN {X 0,Y 387.398,Z 398.139,A -85,B 0,C 180,E1 -11985.253,E2 -11985.253} C_VEL
LIN {X 0,Y 388.058,Z 379.672,A -85,B 0,C 180,E1 -11985.785,E2 -11985.785} C_VEL
LIN {X 0,Y 389.142,Z 343.086,A -85,B 0,C 180,E1 -11986.763,E2 -11986.763} C_VEL
LIN {X 0,Y 387.469,Z 329.425,A -85,B 0,C 180,E1 -11987.288,E2 -11987.288} C_VEL
LIN {X 0,Y 384.304,Z 313.65,A -85,B 0,C 180,E1 -11988.042,E2 -11988.042} C_VEL
LIN {X 0,Y 385.236,Z 296.782,A -85,B 0,C 180,E1 -11991.654,E2 -11991.654} C_VEL
LIN {X 0,Y 385.563,Z 288.982,A -85,B 0,C 180,E1 -11993.358,E2 -11993.358} C_VEL
LIN {X 0,Y 383.675,Z 280.187,A -85,B 0,C 180,E1 -11995.493,E2 -11995.493} C_VEL
LIN {X 0,Y 383.009,Z 277.594,A -85,B 0,C 180,E1 -11996.203,E2 -11996.203} C_VEL
LIN {X 0,Y 382.983,Z 277.595,A -85,B 0,C 180,E1 -11999.702,E2 -11999.702} C_VEL
LIN {X 0,Y 382.962,Z 277.595,A -85,B 0,C 180,E1 -12002.411,E2 -12002.411} C_VEL
LIN {X 0,Y 382.978,Z 277.592,A -85,B 0,C 180,E1 -12005.962,E2 -12005.962} C_VEL
LIN {X 0,Y 382.989,Z 277.59,A -85,B 0,C 180,E1 -12008.604,E2 -12008.604} C_VEL
LIN {X 0,Y 382.973,Z 277.591,A -85,B 0,C 180,E1 -12011.35,E2 -12011.35} C_VEL
LIN {X 0,Y 382.982,Z 277.589,A -85,B 0,C 180,E1 -12014.297,E2 -12014.297} C_VEL
LIN {X 0,Y 382.994,Z 277.588,A -85,B 0,C 180,E1 -12017.234,E2 -12017.234} C_VEL
LIN {X 0,Y 383.003,Z 277.584,A -85,B 0,C 180,E1 -12020.418,E2 -12020.418} C_VEL
LIN {X 0,Y 383.031,Z 277.581,A -85,B 0,C 180,E1 -12024.041,E2 -12024.041} C_VEL
LIN {X 0,Y 383.003,Z 277.588,A -85,B 0,C 180,E1 -12027.576,E2 -12027.576} C_VEL
LIN {X 0,Y 382.995,Z 277.591,A -85,B 0,C 180,E1 -12030.296,E2 -12030.296} C_VEL
LIN {X 0,Y 383.021,Z 277.591,A -85,B 0,C 180,E1 -12034.042,E2 -12034.042} C_VEL
LIN {X 0,Y 383.007,Z 277.593,A -85,B 0,C 180,E1 -12037.331,E2 -12037.331} C_VEL
LIN {X 0,Y 383.086,Z 277.613,A -85,B 0,C 180,E1 -12039.806,E2 -12039.806} C_VEL
LIN {X 0,Y 386.255,Z 288.908,A -85,B 0,C 180,E1 -12042.115,E2 -12042.115} C_VEL
LIN {X 0,Y 387.887,Z 294.967,A -85,B 0,C 180,E1 -12042.437,E2 -12042.437} C_VEL
LIN {X 0,Y 390.057,Z 308.334,A -85,B 0,C 180,E1 -12043.018,E2 -12043.018} C_VEL
LIN {X 0,Y 387.91,Z 371.095,A -85,B 0,C 180,E1 -12044.731,E2 -12044.731} C_VEL
LIN {X 0,Y 387.299,Z 383.069,A -85,B 0,C 180,E1 -12045.278,E2 -12045.278} C_VEL
LIN {X 0,Y 386.717,Z 393.07,A -85,B 0,C 180,E1 -12045.928,E2 -12045.928} C_VEL
LIN {X 0,Y 385.974,Z 403.93,A -85,B 0,C 180,E1 -12046.839,E2 -12046.839} C_VEL
LIN {X 0,Y 385.263,Z 413.391,A -85,B 0,C 180,E1 -12047.886,E2 -12047.886} C_VEL
LIN {X 0,Y 384.586,Z 421.01,A -85,B 0,C 180,E1 -12048.933,E2 -12048.933} C_VEL
LIN {X 0,Y 383.975,Z 427.301,A -85,B 0,C 180,E1 -12049.982,E2 -12049.982} C_VEL
LIN {X 0,Y 383.42,Z 432.534,A -85,B 0,C 180,E1 -12051.032,E2 -12051.032} C_VEL
LIN {X 0,Y 383.069,Z 437.26,A -85,B 0,C 180,E1 -12052.193,E2 -12052.193} C_VEL
LIN {X 0,Y 382.447,Z 442.019,A -85,B 0,C 180,E1 -12053.665,E2 -12053.665} C_VEL
LIN {X 0,Y 382.149,Z 444.583,A -85,B 0,C 180,E1 -12054.719,E2 -12054.719} C_VEL
LIN {X 0,Y 382.167,Z 446.558,A -85,B 0,C 180,E1 -12055.776,E2 -12055.776} C_VEL
LIN {X 0,Y 381.975,Z 448.007,A -85,B 0,C 180,E1 -12056.831,E2 -12056.831} C_VEL
LIN {X 0,Y 381.806,Z 448.919,A -85,B 0,C 180,E1 -12057.885,E2 -12057.885} C_VEL
LIN {X 0,Y 381.687,Z 449.213,A -85,B 0,C 180,E1 -12058.94,E2 -12058.94} C_VEL
LIN {X 0,Y 381.662,Z 448.952,A -85,B 0,C 180,E1 -12059.995,E2 -12059.995} C_VEL
LIN {X 0,Y 381.664,Z 448.183,A -85,B 0,C 180,E1 -12061.05,E2 -12061.05} C_VEL
LIN {X 0,Y 381.686,Z 446.891,A -85,B 0,C 180,E1 -12062.105,E2 -12062.105} C_VEL
LIN {X 0,Y 381.777,Z 443.824,A -85,B 0,C 180,E1 -12063.689,E2 -12063.689} C_VEL
LIN {X 0,Y 381.879,Z 441.033,A -85,B 0,C 180,E1 -12064.745,E2 -12064.745} C_VEL
LIN {X 0,Y 382.037,Z 435.56,A -85,B 0,C 180,E1 -12066.331,E2 -12066.331} C_VEL
LIN {X 0,Y 382.415,Z 428.289,A -85,B 0,C 180,E1 -12067.917,E2 -12067.917} C_VEL
LIN {X 0,Y 382.672,Z 422.145,A -85,B 0,C 180,E1 -12068.975,E2 -12068.975} C_VEL
LIN {X 0,Y 382.966,Z 414.675,A -85,B 0,C 180,E1 -12070.034,E2 -12070.034} C_VEL
LIN {X 0,Y 383.444,Z 406.756,A -85,B 0,C 180,E1 -12070.956,E2 -12070.956} C_VEL
LIN {X 0,Y 383.753,Z 398.443,A -85,B 0,C 180,E1 -12071.75,E2 -12071.75} C_VEL
LIN {X 0,Y 384.152,Z 388.022,A -85,B 0,C 180,E1 -12072.542,E2 -12072.542} C_VEL
LIN {X 0,Y 384.538,Z 376.519,A -85,B 0,C 180,E1 -12073.166,E2 -12073.166} C_VEL
LIN {X 0,Y 384.702,Z 366.928,A -85,B 0,C 180,E1 -12073.53,E2 -12073.53} C_VEL
LIN {X 0,Y 385.61,Z 307.162,A -85,B 0,C 180,E1 -12074.989,E2 -12074.989} C_VEL
LIN {X 0,Y 383.103,Z 289.81,A -85,B 0,C 180,E1 -12075.513,E2 -12075.513} C_VEL
LIN {X 0,Y 383.397,Z 280.78,A -85,B 0,C 180,E1 -12078.151,E2 -12078.151} C_VEL
LIN {X 0,Y 383.129,Z 277.572,A -85,B 0,C 180,E1 -12079.134,E2 -12079.134} C_VEL
LIN {X 0,Y 382.994,Z 277.589,A -85,B 0,C 180,E1 -12083.433,E2 -12083.433} C_VEL
LIN {X 0,Y 382.968,Z 277.594,A -85,B 0,C 180,E1 -12086.124,E2 -12086.124} C_VEL
LIN {X 0,Y 382.957,Z 277.594,A -85,B 0,C 180,E1 -12089.695,E2 -12089.695} C_VEL
LIN {X 0,Y 382.982,Z 277.59,A -85,B 0,C 180,E1 -12093.394,E2 -12093.394} C_VEL
LIN {X 0,Y 383.007,Z 277.59,A -85,B 0,C 180,E1 -12096.158,E2 -12096.158} C_VEL
LIN {X 0,Y 382.95,Z 277.595,A -85,B 0,C 180,E1 -12099.956,E2 -12099.956} C_VEL
LIN {X 0,Y 382.977,Z 277.593,A -85,B 0,C 180,E1 -12102.772,E2 -12102.772} C_VEL
LIN {X 0,Y 382.965,Z 277.592,A -85,B 0,C 180,E1 -12105.783,E2 -12105.783} C_VEL
LIN {X 0,Y 382.953,Z 277.596,A -85,B 0,C 180,E1 -12108.79,E2 -12108.79} C_VEL
LIN {X 0,Y 382.96,Z 277.593,A -85,B 0,C 180,E1 -12112.091,E2 -12112.091} C_VEL
LIN {X 0,Y 382.979,Z 277.594,A -85,B 0,C 180,E1 -12115.326,E2 -12115.326} C_VEL
LIN {X 0,Y 382.94,Z 277.597,A -85,B 0,C 180,E1 -12119.076,E2 -12119.076} C_VEL
LIN {X 0,Y 383.012,Z 277.587,A -85,B 0,C 180,E1 -12122.693,E2 -12122.693} C_VEL
LIN {X 0,Y 383.005,Z 277.59,A -85,B 0,C 180,E1 -12125.035,E2 -12125.035} C_VEL
LIN {X 0,Y 382.944,Z 277.594,A -85,B 0,C 180,E1 -12128.465,E2 -12128.465} C_VEL
LIN {X 0,Y 383.012,Z 277.589,A -85,B 0,C 180,E1 -12131.822,E2 -12131.822} C_VEL
LIN {X 0,Y 383.059,Z 277.582,A -85,B 0,C 180,E1 -12135.115,E2 -12135.115} C_VEL
LIN {X 0,Y 383.055,Z 277.581,A -85,B 0,C 180,E1 -12138.355,E2 -12138.355} C_VEL
LIN {X 0,Y 383.21,Z 277.564,A -85,B 0,C 180,E1 -12141.972,E2 -12141.972} C_VEL
LIN {X 0,Y 383.15,Z 277.569,A -85,B 0,C 180,E1 -12144.736,E2 -12144.736} C_VEL
LIN {X 0,Y 383.335,Z 277.548,A -85,B 0,C 180,E1 -12147.897,E2 -12147.897} C_VEL
LIN {X 0,Y 383.465,Z 277.532,A -85,B 0,C 180,E1 -12149.998,E2 -12149.998} C_VEL
LIN {X 0,Y 383.226,Z 277.559,A -85,B 0,C 180,E1 -12153.152,E2 -12153.152} C_VEL
LIN {X 0,Y 383.227,Z 277.562,A -85,B 0,C 180,E1 -12156.315,E2 -12156.315} C_VEL
LIN {X 0,Y 383.1,Z 277.575,A -85,B 0,C 180,E1 -12159.501,E2 -12159.501} C_VEL
LIN {X 0,Y 383.084,Z 277.58,A -85,B 0,C 180,E1 -12162.716,E2 -12162.716} C_VEL
LIN {X 0,Y 383.022,Z 277.587,A -85,B 0,C 180,E1 -12165.974,E2 -12165.974} C_VEL
LIN {X 0,Y 383.002,Z 277.588,A -85,B 0,C 180,E1 -12169.285,E2 -12169.285} C_VEL
LIN {X 0,Y 382.95,Z 277.596,A -85,B 0,C 180,E1 -12172.651,E2 -12172.651} C_VEL
LIN {X 0,Y 382.338,Z 277.679,A -85,B 0,C 180,E1 -12173.529,E2 -12173.529} C_VEL
LIN {X 0,Y 379.502,Z 278.032,A -85,B 0,C 180,E1 -12174.957,E2 -12174.957} C_VEL
LIN {X 0,Y 377.067,Z 278.33,A -85,B 0,C 180,E1 -12176.112,E2 -12176.112} C_VEL
LIN {X 0,Y 376.019,Z 278.461,A -85,B 0,C 180,E1 -12177.005,E2 -12177.005} C_VEL
LIN {X 0,Y 375.934,Z 278.466,A -85,B 0,C 180,E1 -12177.308,E2 -12177.308} C_VEL
LIN {X 0,Y 375.904,Z 278.474,A -85,B 0,C 180,E1 -12180.696,E2 -12180.696} C_VEL
LIN {X 0,Y 375.907,Z 278.471,A -85,B 0,C 180,E1 -12184.114,E2 -12184.114} C_VEL
LIN {X 0,Y 375.904,Z 278.474,A -85,B 0,C 180,E1 -12186.744,E2 -12186.744} C_VEL
LIN {X 0,Y 375.95,Z 278.466,A -85,B 0,C 180,E1 -12189.976,E2 -12189.976} C_VEL
LIN {X 0,Y 375.953,Z 278.467,A -85,B 0,C 180,E1 -12193.759,E2 -12193.759} C_VEL
LIN {X 0,Y 375.953,Z 278.467,A -85,B 0,C 180,E1 -12196.804,E2 -12196.804} C_VEL
LIN {X 0,Y 375.955,Z 278.466,A -85,B 0,C 180,E1 -12200.032,E2 -12200.032} C_VEL
LIN {X 0,Y 375.923,Z 278.472,A -85,B 0,C 180,E1 -12203.5,E2 -12203.5} C_VEL
LIN {X 0,Y 375.92,Z 278.472,A -85,B 0,C 180,E1 -12205.893,E2 -12205.893} C_VEL
LIN {X 0,Y 375.926,Z 278.472,A -85,B 0,C 180,E1 -12209.692,E2 -12209.692} C_VEL
LIN {X 0,Y 375.984,Z 278.464,A -85,B 0,C 180,E1 -12213.353,E2 -12213.353} C_VEL
LIN {X 0,Y 375.945,Z 278.466,A -85,B 0,C 180,E1 -12216.892,E2 -12216.892} C_VEL
LIN {X 0,Y 375.966,Z 278.466,A -85,B 0,C 180,E1 -12220.344,E2 -12220.344} C_VEL
LIN {X 0,Y 375.997,Z 278.463,A -85,B 0,C 180,E1 -12223.724,E2 -12223.724} C_VEL
LIN {X 0,Y 376.078,Z 278.449,A -85,B 0,C 180,E1 -12227.047,E2 -12227.047} C_VEL
LIN {X 0,Y 376.089,Z 278.452,A -85,B 0,C 180,E1 -12230.324,E2 -12230.324} C_VEL
LIN {X 0,Y 376.205,Z 278.434,A -85,B 0,C 180,E1 -12233.57,E2 -12233.57} C_VEL
LIN {X 0,Y 376.321,Z 278.42,A -85,B 0,C 180,E1 -12237.865,E2 -12237.865} C_VEL
LIN {X 0,Y 376.329,Z 278.421,A -85,B 0,C 180,E1 -12242.146,E2 -12242.146} C_VEL
LIN {X 0,Y 376.186,Z 278.439,A -85,B 0,C 180,E1 -12246.441,E2 -12246.441} C_VEL
LIN {X 0,Y 376.101,Z 278.447,A -85,B 0,C 180,E1 -12249.687,E2 -12249.687} C_VEL
LIN {X 0,Y 376.08,Z 278.449,A -85,B 0,C 180,E1 -12253.663,E2 -12253.663} C_VEL
LIN {X 0,Y 375.999,Z 278.46,A -85,B 0,C 180,E1 -12257.594,E2 -12257.594} C_VEL
LIN {X 0,Y 375.973,Z 278.465,A -85,B 0,C 180,E1 -12260.837,E2 -12260.837} C_VEL
LIN {X 0,Y 375.93,Z 278.468,A -85,B 0,C 180,E1 -12264.29,E2 -12264.29} C_VEL
LIN {X 0,Y 375.922,Z 278.47,A -85,B 0,C 180,E1 -12266.664,E2 -12266.664} C_VEL
LIN {X 0,Y 375.916,Z 278.472,A -85,B 0,C 180,E1 -12269.088,E2 -12269.088} C_VEL
LIN {X 0,Y 375.954,Z 278.469,A -85,B 0,C 180,E1 -12271.567,E2 -12271.567} C_VEL
LIN {X 0,Y 375.947,Z 278.469,A -85,B 0,C 180,E1 -12275.421,E2 -12275.421} C_VEL
LIN {X 0,Y 375.933,Z 278.468,A -85,B 0,C 180,E1 -12278.266,E2 -12278.266} C_VEL
LIN {X 0,Y 375.914,Z 278.473,A -85,B 0,C 180,E1 -12281.601,E2 -12281.601} C_VEL
LIN {X 0,Y 375.92,Z 278.469,A -85,B 0,C 180,E1 -12284.734,E2 -12284.734} C_VEL
LIN {X 0,Y 375.909,Z 278.473,A -85,B 0,C 180,E1 -12287.7,E2 -12287.7} C_VEL
LIN {X 0,Y 375.937,Z 278.468,A -85,B 0,C 180,E1 -12290.537,E2 -12290.537} C_VEL
LIN {X 0,Y 375.961,Z 278.466,A -85,B 0,C 180,E1 -12293.501,E2 -12293.501} C_VEL
LIN {X 0,Y 375.962,Z 278.467,A -85,B 0,C 180,E1 -12295.892,E2 -12295.892} C_VEL
LIN {X 0,Y 375.966,Z 278.465,A -85,B 0,C 180,E1 -12299.69,E2 -12299.69} C_VEL
LIN {X 0,Y 375.931,Z 278.468,A -85,B 0,C 180,E1 -12303.344,E2 -12303.344} C_VEL
LIN {X 0,Y 376.057,Z 278.626,A -85,B 0,C 180,E1 -12304.317,E2 -12304.317} C_VEL
LIN {X 0,Y 377.48,Z 286.676,A -85,B 0,C 180,E1 -12306.478,E2 -12306.478} C_VEL
LIN {X 0,Y 377.599,Z 292.026,A -85,B 0,C 180,E1 -12307.86,E2 -12307.86} C_VEL
LIN {X 0,Y 376.538,Z 306.421,A -85,B 0,C 180,E1 -12311.502,E2 -12311.502} C_VEL
LIN {X 0,Y 375.861,Z 317.596,A -85,B 0,C 180,E1 -12314.306,E2 -12314.306} C_VEL
LIN {X 0,Y 378.443,Z 343.622,A -85,B 0,C 180,E1 -12315.038,E2 -12315.038} C_VEL
LIN {X 0,Y 377.553,Z 396.158,A -85,B 0,C 180,E1 -12316.376,E2 -12316.376} C_VEL
LIN {X 0,Y 377.172,Z 408.132,A -85,B 0,C 180,E1 -12316.876,E2 -12316.876} C_VEL
LIN {X 0,Y 376.72,Z 417.922,A -85,B 0,C 180,E1 -12317.477,E2 -12317.477} C_VEL
LIN {X 0,Y 376.333,Z 426.472,A -85,B 0,C 180,E1 -12318.148,E2 -12318.148} C_VEL
LIN {X 0,Y 375.88,Z 434.747,A -85,B 0,C 180,E1 -12318.953,E2 -12318.953} C_VEL
LIN {X 0,Y 375.595,Z 441.635,A -85,B 0,C 180,E1 -12319.763,E2 -12319.763} C_VEL
LIN {X 0,Y 375.319,Z 447.493,A -85,B 0,C 180,E1 -12320.572,E2 -12320.572} C_VEL
LIN {X 0,Y 375.064,Z 454.043,A -85,B 0,C 180,E1 -12321.652,E2 -12321.652} C_VEL
LIN {X 0,Y 374.876,Z 459.473,A -85,B 0,C 180,E1 -12322.732,E2 -12322.732} C_VEL
LIN {X 0,Y 374.713,Z 463.813,A -85,B 0,C 180,E1 -12323.767,E2 -12323.767} C_VEL
LIN {X 0,Y 374.68,Z 468.487,A -85,B 0,C 180,E1 -12325.16,E2 -12325.16} C_VEL
LIN {X 0,Y 374.534,Z 471.309,A -85,B 0,C 180,E1 -12326.236,E2 -12326.236} C_VEL
LIN {X 0,Y 374.599,Z 474.362,A -85,B 0,C 180,E1 -12327.851,E2 -12327.851} C_VEL
LIN {X 0,Y 374.614,Z 475.657,A -85,B 0,C 180,E1 -12328.927,E2 -12328.927} C_VEL
LIN {X 0,Y 374.594,Z 476.417,A -85,B 0,C 180,E1 -12330.002,E2 -12330.002} C_VEL
LIN {X 0,Y 374.543,Z 476.642,A -85,B 0,C 180,E1 -12331.077,E2 -12331.077} C_VEL
LIN {X 0,Y 374.478,Z 476.238,A -85,B 0,C 180,E1 -12332.153,E2 -12332.153} C_VEL
LIN {X 0,Y 374.48,Z 475.275,A -85,B 0,C 180,E1 -12333.229,E2 -12333.229} C_VEL
LIN {X 0,Y 374.642,Z 472.895,A -85,B 0,C 180,E1 -12334.844,E2 -12334.844} C_VEL
LIN {X 0,Y 374.763,Z 469.169,A -85,B 0,C 180,E1 -12336.462,E2 -12336.462} C_VEL
LIN {X 0,Y 375.014,Z 465.894,A -85,B 0,C 180,E1 -12337.54,E2 -12337.54} C_VEL
LIN {X 0,Y 375.544,Z 459.524,A -85,B 0,C 180,E1 -12339.155,E2 -12339.155} C_VEL
LIN {X 0,Y 376.084,Z 454.263,A -85,B 0,C 180,E1 -12340.228,E2 -12340.228} C_VEL
LIN {X 0,Y 376.71,Z 447.949,A -85,B 0,C 180,E1 -12341.298,E2 -12341.298} C_VEL
LIN {X 0,Y 377.375,Z 440.324,A -85,B 0,C 180,E1 -12342.368,E2 -12342.368} C_VEL
LIN {X 0,Y 378.124,Z 432.287,A -85,B 0,C 180,E1 -12343.299,E2 -12343.299} C_VEL
LIN {X 0,Y 379.038,Z 422.415,A -85,B 0,C 180,E1 -12344.223,E2 -12344.223} C_VEL
LIN {X 0,Y 379.895,Z 411.133,A -85,B 0,C 180,E1 -12345.012,E2 -12345.012} C_VEL
LIN {X 0,Y 380.64,Z 401.05,A -85,B 0,C 180,E1 -12345.53,E2 -12345.53} C_VEL
LIN {X 0,Y 381.29,Z 389.33,A -85,B 0,C 180,E1 -12345.949,E2 -12345.949} C_VEL
LIN {X 0,Y 382.692,Z 343.608,A -85,B 0,C 180,E1 -12347.205,E2 -12347.205} C_VEL
LIN {X 0,Y 381.122,Z 330.674,A -85,B 0,C 180,E1 -12347.735,E2 -12347.735} C_VEL
LIN {X 0,Y 377.768,Z 314.496,A -85,B 0,C 180,E1 -12348.529,E2 -12348.529} C_VEL
LIN {X 0,Y 377.56,Z 313.1,A -85,B 0,C 180,E1 -12348.639,E2 -12348.639} C_VEL
LIN {X 0,Y 378.646,Z 296.096,A -85,B 0,C 180,E1 -12352.366,E2 -12352.366} C_VEL
LIN {X 0,Y 378.829,Z 290.911,A -85,B 0,C 180,E1 -12353.509,E2 -12353.509} C_VEL
LIN {X 0,Y 376.914,Z 282.203,A -85,B 0,C 180,E1 -12355.704,E2 -12355.704} C_VEL
LIN {X 0,Y 375.969,Z 278.472,A -85,B 0,C 180,E1 -12356.733,E2 -12356.733} C_VEL
LIN {X 0,Y 375.968,Z 278.47,A -85,B 0,C 180,E1 -12360.314,E2 -12360.314} C_VEL
LIN {X 0,Y 375.915,Z 278.473,A -85,B 0,C 180,E1 -12364.118,E2 -12364.118} C_VEL
LIN {X 0,Y 375.935,Z 278.469,A -85,B 0,C 180,E1 -12366.745,E2 -12366.745} C_VEL
LIN {X 0,Y 375.952,Z 278.463,A -85,B 0,C 180,E1 -12369.96,E2 -12369.96} C_VEL
LIN {X 0,Y 375.913,Z 278.472,A -85,B 0,C 180,E1 -12373.182,E2 -12373.182} C_VEL
LIN {X 0,Y 375.913,Z 278.473,A -85,B 0,C 180,E1 -12376.816,E2 -12376.816} C_VEL
LIN {X 0,Y 375.952,Z 278.463,A -85,B 0,C 180,E1 -12380.532,E2 -12380.532} C_VEL
LIN {X 0,Y 375.976,Z 278.46,A -85,B 0,C 180,E1 -12383.495,E2 -12383.495} C_VEL
LIN {X 0,Y 375.975,Z 278.462,A -85,B 0,C 180,E1 -12385.886,E2 -12385.886} C_VEL
LIN {X 0,Y 375.979,Z 278.466,A -85,B 0,C 180,E1 -12389.684,E2 -12389.684} C_VEL
LIN {X 0,Y 375.946,Z 278.469,A -85,B 0,C 180,E1 -12392.133,E2 -12392.133} C_VEL
LIN {X 0,Y 375.989,Z 278.469,A -85,B 0,C 180,E1 -12395.714,E2 -12395.714} C_VEL
LIN {X 0,Y 376.015,Z 278.51,A -85,B 0,C 180,E1 -12399.194,E2 -12399.194} C_VEL
LIN {X 0,Y 379.26,Z 289.516,A -85,B 0,C 180,E1 -12401.542,E2 -12401.542} C_VEL
LIN {X 0,Y 381.274,Z 294.682,A -85,B 0,C 180,E1 -12401.883,E2 -12401.883} C_VEL
LIN {X 0,Y 383.75,Z 309.111,A -85,B 0,C 180,E1 -12402.553,E2 -12402.553} C_VEL
LIN {X 0,Y 381.395,Z 371.762,A -85,B 0,C 180,E1 -12404.327,E2 -12404.327} C_VEL
LIN {X 0,Y 380.754,Z 383.57,A -85,B 0,C 180,E1 -12404.883,E2 -12404.883} C_VEL
LIN {X 0,Y 380.132,Z 393.531,A -85,B 0,C 180,E1 -12405.542,E2 -12405.542} C_VEL
LIN {X 0,Y 379.451,Z 402.863,A -85,B 0,C 180,E1 -12406.336,E2 -12406.336} C_VEL
LIN {X 0,Y 378.586,Z 412.701,A -85,B 0,C 180,E1 -12407.396,E2 -12407.396} C_VEL
LIN {X 0,Y 377.914,Z 420.425,A -85,B 0,C 180,E1 -12408.463,E2 -12408.463} C_VEL
LIN {X 0,Y 377.22,Z 426.854,A -85,B 0,C 180,E1 -12409.529,E2 -12409.529} C_VEL
LIN {X 0,Y 376.475,Z 433.413,A -85,B 0,C 180,E1 -12410.865,E2 -12410.865} C_VEL
LIN {X 0,Y 376.058,Z 438.24,A -85,B 0,C 180,E1 -12412.101,E2 -12412.101} C_VEL
LIN {X 0,Y 375.433,Z 442.715,A -85,B 0,C 180,E1 -12413.546,E2 -12413.546} C_VEL
LIN {X 0,Y 375.1,Z 445.186,A -85,B 0,C 180,E1 -12414.619,E2 -12414.619} C_VEL
LIN {X 0,Y 375.101,Z 447.062,A -85,B 0,C 180,E1 -12415.697,E2 -12415.697} C_VEL
LIN {X 0,Y 374.908,Z 448.42,A -85,B 0,C 180,E1 -12416.771,E2 -12416.771} C_VEL
LIN {X 0,Y 374.73,Z 449.265,A -85,B 0,C 180,E1 -12417.845,E2 -12417.845} C_VEL
LIN {X 0,Y 374.623,Z 449.53,A -85,B 0,C 180,E1 -12418.92,E2 -12418.92} C_VEL
LIN {X 0,Y 374.595,Z 449.191,A -85,B 0,C 180,E1 -12419.995,E2 -12419.995} C_VEL
LIN {X 0,Y 374.566,Z 448.339,A -85,B 0,C 180,E1 -12421.07,E2 -12421.07} C_VEL
LIN {X 0,Y 374.587,Z 446.963,A -85,B 0,C 180,E1 -12422.145,E2 -12422.145} C_VEL
LIN {X 0,Y 374.692,Z 443.792,A -85,B 0,C 180,E1 -12423.758,E2 -12423.758} C_VEL
LIN {X 0,Y 374.812,Z 440.903,A -85,B 0,C 180,E1 -12424.835,E2 -12424.835} C_VEL
LIN {X 0,Y 374.902,Z 436.292,A -85,B 0,C 180,E1 -12426.189,E2 -12426.189} C_VEL
LIN {X 0,Y 375.229,Z 430.531,A -85,B 0,C 180,E1 -12427.528,E2 -12427.528} C_VEL
LIN {X 0,Y 375.537,Z 423.229,A -85,B 0,C 180,E1 -12428.876,E2 -12428.876} C_VEL
LIN {X 0,Y 375.888,Z 414.857,A -85,B 0,C 180,E1 -12430.089,E2 -12430.089} C_VEL
LIN {X 0,Y 376.379,Z 406.912,A -85,B 0,C 180,E1 -12431.028,E2 -12431.028} C_VEL
LIN {X 0,Y 376.672,Z 398.564,A -85,B 0,C 180,E1 -12431.837,E2 -12431.837} C_VEL
LIN {X 0,Y 377.112,Z 388.109,A -85,B 0,C 180,E1 -12432.643,E2 -12432.643} C_VEL
LIN {X 0,Y 377.498,Z 376.541,A -85,B 0,C 180,E1 -12433.279,E2 -12433.279} C_VEL
LIN {X 0,Y 377.669,Z 366.948,A -85,B 0,C 180,E1 -12433.65,E2 -12433.65} C_VEL
LIN {X 0,Y 378.528,Z 307.204,A -85,B 0,C 180,E1 -12435.165,E2 -12435.165} C_VEL
LIN {X 0,Y 376.069,Z 290.072,A -85,B 0,C 180,E1 -12435.687,E2 -12435.687} C_VEL
LIN {X 0,Y 376.371,Z 282.049,A -85,B 0,C 180,E1 -12438.059,E2 -12438.059} C_VEL
LIN {X 0,Y 376.1,Z 278.448,A -85,B 0,C 180,E1 -12439.222,E2 -12439.222} C_VEL
LIN {X 0,Y 375.959,Z 278.466,A -85,B 0,C 180,E1 -12443.652,E2 -12443.652} C_VEL
LIN {X 0,Y 375.897,Z 278.475,A -85,B 0,C 180,E1 -12446.654,E2 -12446.654} C_VEL
LIN {X 0,Y 375.896,Z 278.473,A -85,B 0,C 180,E1 -12449.077,E2 -12449.077} C_VEL
LIN {X 0,Y 375.92,Z 278.469,A -85,B 0,C 180,E1 -12451.557,E2 -12451.557} C_VEL
LIN {X 0,Y 375.958,Z 278.468,A -85,B 0,C 180,E1 -12454.661,E2 -12454.661} C_VEL
LIN {X 0,Y 375.911,Z 278.474,A -85,B 0,C 180,E1 -12458.256,E2 -12458.256} C_VEL
LIN {X 0,Y 375.892,Z 278.473,A -85,B 0,C 180,E1 -12461.592,E2 -12461.592} C_VEL
LIN {X 0,Y 375.895,Z 278.475,A -85,B 0,C 180,E1 -12464.725,E2 -12464.725} C_VEL
LIN {X 0,Y 375.9,Z 278.474,A -85,B 0,C 180,E1 -12468.393,E2 -12468.393} C_VEL
LIN {X 0,Y 375.933,Z 278.468,A -85,B 0,C 180,E1 -12471.725,E2 -12471.725} C_VEL
LIN {X 0,Y 375.941,Z 278.47,A -85,B 0,C 180,E1 -12475.327,E2 -12475.327} C_VEL
LIN {X 0,Y 375.915,Z 278.47,A -85,B 0,C 180,E1 -12478.432,E2 -12478.432} C_VEL
LIN {X 0,Y 375.938,Z 278.467,A -85,B 0,C 180,E1 -12482.135,E2 -12482.135} C_VEL
LIN {X 0,Y 375.96,Z 278.465,A -85,B 0,C 180,E1 -12484.534,E2 -12484.534} C_VEL
LIN {X 0,Y 375.914,Z 278.471,A -85,B 0,C 180,E1 -12488.041,E2 -12488.041} C_VEL
LIN {X 0,Y 375.958,Z 278.467,A -85,B 0,C 180,E1 -12491.469,E2 -12491.469} C_VEL
LIN {X 0,Y 376.007,Z 278.459,A -85,B 0,C 180,E1 -12494.829,E2 -12494.829} C_VEL
LIN {X 0,Y 376.007,Z 278.46,A -85,B 0,C 180,E1 -12498.134,E2 -12498.134} C_VEL
LIN {X 0,Y 376.166,Z 278.442,A -85,B 0,C 180,E1 -12501.915,E2 -12501.915} C_VEL
LIN {X 0,Y 376.122,Z 278.444,A -85,B 0,C 180,E1 -12504.637,E2 -12504.637} C_VEL
LIN {X 0,Y 376.302,Z 278.424,A -85,B 0,C 180,E1 -12507.858,E2 -12507.858} C_VEL
LIN {X 0,Y 376.434,Z 278.408,A -85,B 0,C 180,E1 -12509.998,E2 -12509.998} C_VEL
LIN {X 0,Y 376.162,Z 278.439,A -85,B 0,C 180,E1 -12513.211,E2 -12513.211} C_VEL
LIN {X 0,Y 376.185,Z 278.44,A -85,B 0,C 180,E1 -12516.434,E2 -12516.434} C_VEL
LIN {X 0,Y 376.067,Z 278.452,A -85,B 0,C 180,E1 -12519.681,E2 -12519.681} C_VEL
LIN {X 0,Y 376.033,Z 278.456,A -85,B 0,C 180,E1 -12523.658,E2 -12523.658} C_VEL
LIN {X 0,Y 375.985,Z 278.461,A -85,B 0,C 180,E1 -12527.607,E2 -12527.607} C_VEL
LIN {X 0,Y 375.922,Z 278.473,A -85,B 0,C 180,E1 -12530.833,E2 -12530.833} C_VEL
LIN {X 0,Y 375.938,Z 278.47,A -85,B 0,C 180,E1 -12534.283,E2 -12534.283} C_VEL
LIN {X 0,Y 375.934,Z 278.466,A -85,B 0,C 180,E1 -12537.308,E2 -12537.308} C_VEL
LIN {X 0,Y 375.258,Z 278.554,A -85,B 0,C 180,E1 -12538.201,E2 -12538.201} C_VEL
LIN {X 0,Y 372.365,Z 278.912,A -85,B 0,C 180,E1 -12539.653,E2 -12539.653} C_VEL
LIN {X 0,Y 369.93,Z 279.219,A -85,B 0,C 180,E1 -12540.827,E2 -12540.827} C_VEL
LIN {X 0,Y 368.907,Z 279.343,A -85,B 0,C 180,E1 -12541.736,E2 -12541.736} C_VEL
LIN {X 0,Y 368.836,Z 279.351,A -85,B 0,C 180,E1 -12542.043,E2 -12542.043} C_VEL
LIN {X 0,Y 368.877,Z 279.35,A -85,B 0,C 180,E1 -12545.004,E2 -12545.004} C_VEL
LIN {X 0,Y 368.863,Z 279.35,A -85,B 0,C 180,E1 -12548.644,E2 -12548.644} C_VEL
LIN {X 0,Y 368.893,Z 279.344,A -85,B 0,C 180,E1 -12552.023,E2 -12552.023} C_VEL
LIN {X 0,Y 368.944,Z 279.341,A -85,B 0,C 180,E1 -12555.197,E2 -12555.197} C_VEL
LIN {X 0,Y 368.896,Z 279.344,A -85,B 0,C 180,E1 -12558.19,E2 -12558.19} C_VEL
LIN {X 0,Y 368.87,Z 279.351,A -85,B 0,C 180,E1 -12561.363,E2 -12561.363} C_VEL
LIN {X 0,Y 368.896,Z 279.347,A -85,B 0,C 180,E1 -12565.151,E2 -12565.151} C_VEL
LIN {X 0,Y 368.892,Z 279.346,A -85,B 0,C 180,E1 -12569.051,E2 -12569.051} C_VEL
LIN {X 0,Y 368.927,Z 279.34,A -85,B 0,C 180,E1 -12572.802,E2 -12572.802} C_VEL
LIN {X 0,Y 368.899,Z 279.347,A -85,B 0,C 180,E1 -12576.123,E2 -12576.123} C_VEL
LIN {X 0,Y 368.899,Z 279.347,A -85,B 0,C 180,E1 -12579.952,E2 -12579.952} C_VEL
LIN {X 0,Y 368.94,Z 279.339,A -85,B 0,C 180,E1 -12583.404,E2 -12583.404} C_VEL
LIN {X 0,Y 369.032,Z 279.328,A -85,B 0,C 180,E1 -12586.796,E2 -12586.796} C_VEL
LIN {X 0,Y 369.039,Z 279.329,A -85,B 0,C 180,E1 -12590.137,E2 -12590.137} C_VEL
LIN {X 0,Y 369.164,Z 279.311,A -85,B 0,C 180,E1 -12593.447,E2 -12593.447} C_VEL
LIN {X 0,Y 369.285,Z 279.296,A -85,B 0,C 180,E1 -12597.824,E2 -12597.824} C_VEL
LIN {X 0,Y 369.188,Z 279.309,A -85,B 0,C 180,E1 -12601.096,E2 -12601.096} C_VEL
LIN {X 0,Y 369.293,Z 279.297,A -85,B 0,C 180,E1 -12602.187,E2 -12602.187} C_VEL
LIN {X 0,Y 369.146,Z 279.316,A -85,B 0,C 180,E1 -12606.564,E2 -12606.564} C_VEL
LIN {X 0,Y 369.051,Z 279.325,A -85,B 0,C 180,E1 -12609.874,E2 -12609.874} C_VEL
LIN {X 0,Y 369.028,Z 279.327,A -85,B 0,C 180,E1 -12613.777,E2 -12613.777} C_VEL
LIN {X 0,Y 368.946,Z 279.338,A -85,B 0,C 180,E1 -12617.75,E2 -12617.75} C_VEL
LIN {X 0,Y 368.903,Z 279.347,A -85,B 0,C 180,E1 -12621.226,E2 -12621.226} C_VEL
LIN {X 0,Y 368.903,Z 279.344,A -85,B 0,C 180,E1 -12623.879,E2 -12623.879} C_VEL
LIN {X 0,Y 368.867,Z 279.351,A -85,B 0,C 180,E1 -12627.216,E2 -12627.216} C_VEL
LIN {X 0,Y 368.893,Z 279.347,A -85,B 0,C 180,E1 -12629.697,E2 -12629.697} C_VEL
LIN {X 0,Y 368.894,Z 279.347,A -85,B 0,C 180,E1 -12633.047,E2 -12633.047} C_VEL
LIN {X 0,Y 368.91,Z 279.343,A -85,B 0,C 180,E1 -12636.202,E2 -12636.202} C_VEL
LIN {X 0,Y 368.873,Z 279.348,A -85,B 0,C 180,E1 -12638.961,E2 -12638.961} C_VEL
LIN {X 0,Y 368.859,Z 279.352,A -85,B 0,C 180,E1 -12642.009,E2 -12642.009} C_VEL
LIN {X 0,Y 368.873,Z 279.348,A -85,B 0,C 180,E1 -12645.178,E2 -12645.178} C_VEL
LIN {X 0,Y 368.862,Z 279.351,A -85,B 0,C 180,E1 -12648.178,E2 -12648.178} C_VEL
LIN {X 0,Y 368.88,Z 279.347,A -85,B 0,C 180,E1 -12651.37,E2 -12651.37} C_VEL
LIN {X 0,Y 368.935,Z 279.339,A -85,B 0,C 180,E1 -12655.149,E2 -12655.149} C_VEL
LIN {X 0,Y 368.902,Z 279.343,A -85,B 0,C 180,E1 -12659.047,E2 -12659.047} C_VEL
LIN {X 0,Y 368.913,Z 279.343,A -85,B 0,C 180,E1 -12661.561,E2 -12661.561} C_VEL
LIN {X 0,Y 369.024,Z 279.468,A -85,B 0,C 180,E1 -12664.214,E2 -12664.214} C_VEL
LIN {X 0,Y 370.607,Z 289.07,A -85,B 0,C 180,E1 -12666.83,E2 -12666.83} C_VEL
LIN {X 0,Y 370.349,Z 295.178,A -85,B 0,C 180,E1 -12668.419,E2 -12668.419} C_VEL
LIN {X 0,Y 369.412,Z 307.916,A -85,B 0,C 180,E1 -12671.699,E2 -12671.699} C_VEL
LIN {X 0,Y 368.815,Z 317.661,A -85,B 0,C 180,E1 -12674.14,E2 -12674.14} C_VEL
LIN {X 0,Y 371.387,Z 344.549,A -85,B 0,C 180,E1 -12674.917,E2 -12674.917} C_VEL
